// TwinCAT 3 PLC project plcProg
// ProgramVersion: 3.1.4024.0
// libraries:
//   Tc2_Standard, * (Beckhoff Automation GmbH)
//   Tc2_System, * (Beckhoff Automation GmbH)
//   Tc2_Utilities, * (Beckhoff Automation GmbH)
//   Tc3_Module, * (Beckhoff Automation GmbH)
//   VisuSymbols,3.5.10.0,System
// project tree:
//   DUTs/ E_EventType.TcDUT, E_OutputLevel.TcDUT, E_Direction.TcDUT, ST_Event.TcDUT
//   / GlobalTextList.TcGTLO, PlcTask.TcTTO, Visualization Manager.TcVMO (not stored)
//   GVLs/ GVL.TcGVL, HMI.TcGVL
//   POUs/ GroupController.TcPOU, SequentialLightSwitch.TcPOU, MAIN.TcPOU, ShutterSwitch.TcPOU, SimpleButton.TcPOU, UpStopDownButton.TcPOU
//   POUs/log_persistence/ EventLogger.TcPOU, FB_CsvPersistentEventStorage.TcPOU, F_UpdateEventTimestampWithSystemTime.TcPOU, I_PersistentEventStorage.TcIO (not stored)
//   VISUs/ Screen1.TcVIS
// real-time tasks:
//   TASK PlcTask: cycle T#10ms, priority 20, ADS port 350
// I/O:
//   DEVICE Device 1 (Beckhoff CCAT)
//   DEVICE Device 2 (CX-BK)
//     Box 1 (CX-BK)
// variable links:
//   plcProg/plcProg Instance <-> Device 2 (CX-BK)/Box 1 (CX-BK)
//     PlcTask Inputs/GVL.din_01zModulu3_przewod_14_s_26_1_gabinetNajnizej_bialopomaranczowy <-> Term 4 (KL1809)/Channel 1/Input
//     PlcTask Inputs/GVL.din_01zModulu4_przewod_11_s_42_1_rodzicow_1z1_bialobrazowy <-> Term 5 (KL1809)/Channel 1/Input
//     PlcTask Inputs/GVL.din_02zModulu3_przewod_14_s_26_1_gabinet_2z2_niebieski <-> Term 4 (KL1809)/Channel 2/Input
//     PlcTask Inputs/GVL.din_02zModulu4_przewod_11_s_42_1_rodzicow_1z1_bialopomaranczowy <-> Term 5 (KL1809)/Channel 2/Input
//     PlcTask Inputs/GVL.din_03zModulu2_przewod_3_s_30_1_kuchnia_2z2_zielony <-> Term 3 (KL1809)/Channel 3/Input
//     PlcTask Inputs/GVL.din_03zModulu3_przewod_14_s_26_1_gabinet_1z2_pomaranczowy <-> Term 4 (KL1809)/Channel 3/Input
//     PlcTask Inputs/GVL.din_03zModulu4_przewod_11_s_42_1_rodzicow_1z2_bialoniebieski <-> Term 5 (KL1809)/Channel 3/Input
//     PlcTask Inputs/GVL.din_04zModulu1_przewod_5_s_27_1_pralnia_2z2_niebieski <-> Term 2 (KL1809)/Channel 4/Input
//     PlcTask Inputs/GVL.din_04zModulu2_przewod_3_s_30_1_kuchnia_1z2_niebieski <-> Term 3 (KL1809)/Channel 4/Input
//     PlcTask Inputs/GVL.din_04zModulu3_przewod_14_s_40_1_lazienka_1z2_zielony <-> Term 4 (KL1809)/Channel 4/Input
//     PlcTask Inputs/GVL.din_05zModulu1_przewod_5_s_27_1_pralnia_1z2_pomaranczowy <-> Term 2 (KL1809)/Channel 5/Input
//     PlcTask Inputs/GVL.din_05zModulu2_przewod_3_s_30_1_kuchnia_2z2_pomaranczowy <-> Term 3 (KL1809)/Channel 5/Input
//     PlcTask Inputs/GVL.din_05zModulu3_przewod_14_s_40_1_lazienka_2z2_niebieski <-> Term 4 (KL1809)/Channel 5/Input
//     PlcTask Inputs/GVL.din_06zModulu1_przewod_1_s_25_1_koniecPrzedpokoju_2z2_zielony <-> Term 2 (KL1809)/Channel 6/Input
//     PlcTask Inputs/GVL.din_06zModulu2_przewod_3_s_30_1_kuchnia_1z2_brazowy <-> Term 3 (KL1809)/Channel 6/Input
//     PlcTask Inputs/GVL.din_07zModulu1_przewod_1_s_5_1_przedpokojPrzyDrzwiach_1z3_niebieski <-> Term 2 (KL1809)/Channel 7/Input
//     PlcTask Inputs/GVL.din_07zModulu2_przewod_3_s_30_1_kuchnia_2z2_bialoniebieski <-> Term 3 (KL1809)/Channel 7/Input
//     PlcTask Inputs/GVL.din_07zModulu3_przewod_5_s_23_1_pralniaNajnizej_niebieski <-> Term 4 (KL1809)/Channel 7/Input
//     PlcTask Inputs/GVL.din_08zModulu1_przewod_1_s_5_1_przedpokojPrzyDrzwiach_2z3_pomaranczowy <-> Term 2 (KL1809)/Channel 8/Input
//     PlcTask Inputs/GVL.din_08zModulu2_przewod_3_s_30_1_kuchnia_1z2_bialopomaranczowy <-> Term 3 (KL1809)/Channel 8/Input
//     PlcTask Inputs/GVL.din_08zModulu3_przewod_13_s_48_1_bezBalkonu_1z2_brazowy <-> Term 4 (KL1809)/Channel 8/Input
//     PlcTask Inputs/GVL.din_09zModulu1_przewod_1_s_5_1_przedpokojPrzyDrzwiach_3z3_brazowy <-> Term 2 (KL1809)/Channel 9/Input
//     PlcTask Inputs/GVL.din_09zModulu3_przewod_13_s_48_1_bezBalkonu_2z2_pomaranczowy <-> Term 4 (KL1809)/Channel 9/Input
//     PlcTask Inputs/GVL.din_10zModulu1_przewod_1_s_25_1_koniecPrzedpokojuElektronicznyPoczworny_1z4_brazowy <-> Term 2 (KL1809)/Channel 10/Input
//     PlcTask Inputs/GVL.din_10zModulu3_przewod_13_s_44_1_bezBalkonu_niebieski <-> Term 4 (KL1809)/Channel 10/Input
//     PlcTask Inputs/GVL.din_11zModulu1_przewod_1_s_25_1_koniecPrzedpokojuElektronicznyPoczworny_2z4_bialoniebieski <-> Term 2 (KL1809)/Channel 11/Input
//     PlcTask Inputs/GVL.din_11zModulu3_przewod_12_s_50_1_zBalkonem_1z2_brazowy <-> Term 4 (KL1809)/Channel 11/Input
//     PlcTask Inputs/GVL.din_12zModulu1_przewod_1_s_25_1_koniecPrzedpokojuElektronicznyPoczworny_3z4_bialopomaranczowy <-> Term 2 (KL1809)/Channel 12/Input
//     PlcTask Inputs/GVL.din_12zModulu2_przewod_4_s_14_1_dolSchodow_2z4_niebieski <-> Term 3 (KL1809)/Channel 12/Input
//     PlcTask Inputs/GVL.din_12zModulu3_przewod_12_s_50_1_zBalkonem_2z2_pomaranczowy <-> Term 4 (KL1809)/Channel 12/Input
//     PlcTask Inputs/GVL.din_13zModulu1_przewod_1_s_25_1_koniecPrzedpokojuElektronicznyPoczworny_4z4_bialobrazowy <-> Term 2 (KL1809)/Channel 13/Input
//     PlcTask Inputs/GVL.din_13zModulu2_przewod_4_s_14_1_dolSchodow_4z4_bialopomaranczowy <-> Term 3 (KL1809)/Channel 13/Input
//     PlcTask Inputs/GVL.din_13zModulu3_przewod_18_s_55_1_korytarzPrzySypialniach_1z1_zielony <-> Term 4 (KL1809)/Channel 13/Input
//     PlcTask Inputs/GVL.din_14ZModulu3_przewod_11_S_42_1_rodzicow_1z2_brazowy <-> Term 4 (KL1809)/Channel 14/Input
//     PlcTask Inputs/GVL.din_14zModulu1_przewod_4_s_21_1_slupekKuchnia_4z4_brazowy <-> Term 2 (KL1809)/Channel 14/Input
//     PlcTask Inputs/GVL.din_14zModulu2_przewod_18_s_38_1_goraSchodow_2z4_pomaranczowy <-> Term 3 (KL1809)/Channel 14/Input
//     PlcTask Inputs/GVL.din_15ZModulu3_przewod_11_S_42_1_rodzicow_2z2_pomaranczowy <-> Term 4 (KL1809)/Channel 15/Input
//     PlcTask Inputs/GVL.din_15zModulu1_przewod_4_s_21_1_slupekKuchnia_1z4_pomaranczowy <-> Term 2 (KL1809)/Channel 15/Input
//     PlcTask Inputs/GVL.din_15zModulu2_przewod_18_s_38_1_goraSchodow_3z4_brazowy <-> Term 3 (KL1809)/Channel 15/Input
//     PlcTask Inputs/GVL.din_16zModulu1_przewod_4_s_21_1_slupekKuchnia_2z4_bialoniebieski <-> Term 2 (KL1809)/Channel 16/Input
//     PlcTask Inputs/GVL.din_16zModulu2_przewod_14_s_26_1_gabinetPrawieNajnizej_brazowy <-> Term 3 (KL1809)/Channel 16/Input
//     PlcTask Inputs/GVL.din_16zModulu3_przewod_11_s_42_1_rodzicow_2z2_niebieski <-> Term 4 (KL1809)/Channel 16/Input
//     PlcTask Inputs/GVL.din_1_1_1 <-> Term 2 (KL1809)/Channel 1/Input
//     PlcTask Inputs/GVL.din_1_2_2 <-> Term 2 (KL1809)/Channel 2/Input
//     PlcTask Outputs/GVL.dout_10_zaluzja_gabinet_w_dol <-> Term 13 (KL2809)/Channel 4/Output
//     PlcTask Outputs/GVL.dout_10zModulu1_przewod_3_o_3_1_swiatloKontuarKuchnia <-> Term 9 (KL2809)/Channel 10/Output
//     PlcTask Outputs/GVL.dout_10zModulu2_przewod_xxx_swiatloGornaLazienkaPodlogowe <-> Term 10 (KL2809)/Channel 10/Output
//     PlcTask Outputs/GVL.dout_11_zaluzja_balkon_w_gore <-> Term 13 (KL2809)/Channel 5/Output
//     PlcTask Outputs/GVL.dout_11zModulu1_przewod_3_o_2_1_swiatloKuchniaSufit <-> Term 9 (KL2809)/Channel 11/Output
//     PlcTask Outputs/GVL.dout_11zModulu2_przewod_13_o_19_1_swiatloSypialniaBezBalkonu <-> Term 10 (KL2809)/Channel 11/Output
//     PlcTask Outputs/GVL.dout_12_zaluzja_balkon_w_dol <-> Term 13 (KL2809)/Channel 6/Output
//     PlcTask Outputs/GVL.dout_12zModulu1_przewod_11_o_18_1_2_swiatloNiskiIWysokiSufitSypialniaRodzicow <-> Term 9 (KL2809)/Channel 12/Output
//     PlcTask Outputs/GVL.dout_13_zaluzja_nad_wykuszem_w_gore <-> Term 13 (KL2809)/Channel 7/Output
//     PlcTask Outputs/GVL.dout_13zModulu1_przewod_4_o_10_1_swiatloGabinet <-> Term 9 (KL2809)/Channel 13/Output
//     PlcTask Outputs/GVL.dout_14_zaluzja_nad_wykuszem_w_dol <-> Term 13 (KL2809)/Channel 8/Output
//     PlcTask Outputs/GVL.dout_14zModulu1_przewod_14_o_24_1_3_swiatloWiszaceGornaLazienka <-> Term 9 (KL2809)/Channel 14/Output
//     PlcTask Outputs/GVL.dout_15_zaluzja_okno_bez_balkonu_w_gore <-> Term 13 (KL2809)/Channel 9/Output
//     PlcTask Outputs/GVL.dout_15zModulu1_przewod_18_o_18_1_2_swiatloKorytarzPunktySufit <-> Term 9 (KL2809)/Channel 15/Output
//     PlcTask Outputs/GVL.dout_16_zaluzja_okno_bez_balkonu_w_dol <-> Term 13 (KL2809)/Channel 10/Output
//     PlcTask Outputs/GVL.dout_16zModulu1_przewod_18_o_18_1_3_swiatloZyrandolKorytarz <-> Term 9 (KL2809)/Channel 16/Output
//     PlcTask Outputs/GVL.dout_1_zaluzja_pralnia_w_gore <-> Term 12 (KL2809)/Channel 11/Output
//     PlcTask Outputs/GVL.dout_1zModulu1_przewod_2_o_4_1_swiatloSalonJadalniaSufit <-> Term 9 (KL2809)/Channel 1/Output
//     PlcTask Outputs/GVL.dout_1zModulu2_przewod_1_s_70_1_swiatloPrzedpokojBlizejSalonu <-> Term 10 (KL2809)/Channel 1/Output
//     PlcTask Outputs/GVL.dout_2_zaluzja_pralnia_w_dol <-> Term 12 (KL2809)/Channel 12/Output
//     PlcTask Outputs/GVL.dout_2zModulu1_przewod_2_o_5_1_swiatloSalonKanapaSufit <-> Term 9 (KL2809)/Channel 2/Output
//     PlcTask Outputs/GVL.dout_2zModulu2_przewod_11_o_17_1_swiatloNadLozkiemSypialniaRodzicow <-> Term 10 (KL2809)/Channel 2/Output
//     PlcTask Outputs/GVL.dout_3_zaluzja_okno_narozne_kuchnia_w_gore <-> Term 12 (KL2809)/Channel 13/Output
//     PlcTask Outputs/GVL.dout_3zModulu1_przewod_2_o_7_1_swiatloPrzejscieZPrzedpokojuDoSalonuSufit <-> Term 9 (KL2809)/Channel 3/Output
//     PlcTask Outputs/GVL.dout_3zModulu2_przewod_14_o_23_1_3_swiatloSlabeGornaLazienka <-> Term 10 (KL2809)/Channel 3/Output
//     PlcTask Outputs/GVL.dout_4_zaluzja_okno_narozne_kuchnia_w_dol <-> Term 12 (KL2809)/Channel 14/Output
//     PlcTask Outputs/GVL.dout_4zModulu2_przewod_14_o_24_1_2_swiatloSrednieGornaLazienka <-> Term 10 (KL2809)/Channel 4/Output
//     PlcTask Outputs/GVL.dout_5_zaluzja_wykusz_w_gore <-> Term 12 (KL2809)/Channel 15/Output
//     PlcTask Outputs/GVL.dout_5zModulu2_przewod_14_o_23_1_2_swiatloMocneGornaLazienka <-> Term 10 (KL2809)/Channel 5/Output
//     PlcTask Outputs/GVL.dout_6_zaluzja_wykusz_w_dol <-> Term 12 (KL2809)/Channel 16/Output
//     PlcTask Outputs/GVL.dout_6zModulu1_przewod_podbitki <-> Term 9 (KL2809)/Channel 6/Output
//     PlcTask Outputs/GVL.dout_6zModulu2_przewod_3_o_1_1_swiatloKuchniaPodSzafkami <-> Term 10 (KL2809)/Channel 6/Output
//     PlcTask Outputs/GVL.dout_7_zaluzja_slide_w_gore <-> Term 13 (KL2809)/Channel 1/Output
//     PlcTask Outputs/GVL.dout_7zModulu1_przewod_1_o_27_1_swiatloPrzedpokojBlizejDrzwi <-> Term 9 (KL2809)/Channel 7/Output
//     PlcTask Outputs/GVL.dout_7zModulu2_przewod_xxxxxx_swiatloTrepy <-> Term 10 (KL2809)/Channel 7/Output
//     PlcTask Outputs/GVL.dout_8_zaluzja_slide_w_dol <-> Term 13 (KL2809)/Channel 2/Output
//     PlcTask Outputs/GVL.dout_8zModulu1_przewod_11_o_18_1_3_swiatloToaletkaSypialniaRodzicow <-> Term 9 (KL2809)/Channel 8/Output
//     PlcTask Outputs/GVL.dout_8zModulu2_przewod_18_o_14_1_swiatloKorytarzPrzypodlogowe <-> Term 10 (KL2809)/Channel 8/Output
//     PlcTask Outputs/GVL.dout_9_zaluzja_gabinet_w_gore <-> Term 13 (KL2809)/Channel 3/Output
//     PlcTask Outputs/GVL.dout_9zModulu1_przewod_5_o_11_1_swiatloPralnia <-> Term 9 (KL2809)/Channel 9/Output

CONFIGURATION plcProg
    RESOURCE PLC ON TwinCAT3
        TASK PlcTask(INTERVAL := T#10ms, PRIORITY := 20);
        PROGRAM MAIN WITH PlcTask : MAIN;
    END_RESOURCE
END_CONFIGURATION

// ---- DUTs/E_EventType.TcDUT
{attribute 'qualified_only'}
{attribute 'strict'}
{attribute 'to_string'}
TYPE E_EventType :
(
	Alarm := 0,
	Message := 1
);
END_TYPE

// ---- DUTs/E_OutputLevel.TcDUT
{attribute 'qualified_only'}
{attribute 'strict'}
{attribute 'to_string'}
TYPE E_OutputLevel :
(
	SMALL := 1,
	MEDIUM := 2,
	BIG := 3,
	SUPERSTRONG := 4	
);
END_TYPE

// ---- DUTs/E_Direction.TcDUT
{attribute 'qualified_only'}
{attribute 'strict'}
{attribute 'to_string'}
TYPE E_Direction :
(
	STOP := 0,
	UP := 1,
	DOWN := 2
);
END_TYPE

// ---- DUTs/ST_Event.TcDUT
TYPE ST_Event :
STRUCT
	eEventType : E_EventType;
	eEventSeverity : TcEventSeverity;
	nEventIdentity : UDINT;
	sEventText : STRING(255);
	dtTimestamp : DATE_AND_TIME;
END_STRUCT
END_TYPE

// ---- GVLs/GVL.TcGVL
{attribute 'qualified_only'}
VAR_GLOBAL CONSTANT
    MAX_SHUTTER_OUTPUTS : INT := 1;
	MAX_LIGHT_OUTPUTS_PER_LEVEL : INT := 3;
	MAX_SIMPLE_OUTPUTS : INT := 3;
	
	MAX_SHUTTERS : INT := 11;
	MAX_SEQUENTIAL_SWITCHES : INT := 0;//TODO 50 ALBO MNIEJ;
	MAX_SIMPLE_BUTTONS : INT := 18; //TODO PEWNIE WIECEJ
END_VAR

VAR_GLOBAL
	
	din_1_1_1 AT %I* : BOOL; //garaż po prawej stronie od drzwi
	din_1_2_2 AT %I* : BOOL; //garaż po lewej stronie od drzwi (wh-gn->bl) + pralnia po lewej stronie od drzwi, pierwszy od dołu (trzeba namierzyć)
	din_1_3_3 AT %I* : BOOL; //pralnia po lewej stronie od drzwi, drugi od dołu (trzeba namierzyć)
	din_1_4_4 AT %I* : BOOL; 
	din_1_5_5 AT %I* : BOOL;
	din_1_6_6 AT %I* : BOOL; 
	din_1_7_7 AT %I* : BOOL;
	din_1_8_8 AT %I* : BOOL;
	din_1_9_9 AT %I* : BOOL; 
	
	din_04zModulu1_przewod_5_s_27_1_pralnia_2z2_niebieski AT %I* : BOOL; //zasilanie bialo-zielony: Wlacznik roletowy w pralni dol
	din_05zModulu1_przewod_5_s_27_1_pralnia_1z2_pomaranczowy AT %I* : BOOL; //zasilanie bialo-zielony: Wlacznik roletowy w pralni gora
	din_06zModulu1_przewod_1_s_25_1_koniecPrzedpokoju_2z2_zielony AT %I* : BOOL; //zasilanie bialo-zielony: Wlacznik podwojny na koncu przedpokoju lub wlacznik poczworny na dole schodow 1/4
	din_07zModulu1_przewod_1_s_5_1_przedpokojPrzyDrzwiach_1z3_niebieski AT %I* : BOOL; //zasilanie bialo-zielony: Wlacznik swiatla w przedpokoju przy drzwiach 1/3
	din_08zModulu1_przewod_1_s_5_1_przedpokojPrzyDrzwiach_2z3_pomaranczowy AT %I* : BOOL; //zasilanie bialo-zielony: Wlacznik swiatla w przedpokoju przy drzwiach 2/3
	din_09zModulu1_przewod_1_s_5_1_przedpokojPrzyDrzwiach_3z3_brazowy AT %I* : BOOL; //zasilanie bialo-zielony: Wlacznik swiatla w przedpokoju przy drzwiach 3/3 lub wlacznik podwojny na koncu przedpokoju 1/2

	din_10zModulu1_przewod_1_s_25_1_koniecPrzedpokojuElektronicznyPoczworny_1z4_brazowy AT %I* : BOOL;//bylo din1_10_10 //zasilanie biało-zielony: Elektroniczny wlacznik swiatla w przedpokoju 1/4 lub wlacznik poczworny w kuchni na slupku 1/4
	din_11zModulu1_przewod_1_s_25_1_koniecPrzedpokojuElektronicznyPoczworny_2z4_bialoniebieski AT %I* : BOOL; //bylo din1_11_11 //zasilanie biało-zielony: Elektroniczny wlacznik swiatla w przedpokoju 2/4
	din_12zModulu1_przewod_1_s_25_1_koniecPrzedpokojuElektronicznyPoczworny_3z4_bialopomaranczowy AT %I* : BOOL; //bylo din1_12_12 //zasilanie biało-zielony: Elektroniczny wlacznik swiatla w przedpokoju 3/4 lub wlacznik poczworny na dole schodow 3/4
	din_13zModulu1_przewod_1_s_25_1_koniecPrzedpokojuElektronicznyPoczworny_4z4_bialobrazowy AT %I* : BOOL; //din_1_13_13 //zasilanie bialo-zielony: Elektroniczny wlacznik swiatla w przedpokoju 4/4	
	
	din_14zModulu1_przewod_4_s_21_1_slupekKuchnia_4z4_brazowy AT %I* : BOOL; //zasilanie bialo-zielony: Wlacznik poczworny w kuchni na slupku 4/4
	din_15zModulu1_przewod_4_s_21_1_slupekKuchnia_1z4_pomaranczowy AT %I* : BOOL; //zasilanie bialo-zielony: Wlacznik poczworny w kuchni na slupku 1/4
	din_16zModulu1_przewod_4_s_21_1_slupekKuchnia_2z4_bialoniebieski AT %I* : BOOL; //zasilanie bialo-zielony: Wlacznik poczworny w kuchni na slupku 2/4

	//todo swiatlo kontuar led, swiatlo zewnetrzne nad drzwiami
	din_03zModulu2_przewod_3_s_30_1_kuchnia_2z2_zielony AT %I* : BOOL; //zasilanie bialo-zielony: Wlacznik roletowy w kuchni kuchnia gora
    din_04zModulu2_przewod_3_s_30_1_kuchnia_1z2_niebieski AT %I* : BOOL; //zasilanie bialo-zielony: Wlacznik roletowy w kuchni kuchnia dol

	din_05zModulu2_przewod_3_s_30_1_kuchnia_2z2_pomaranczowy AT %I* : BOOL; //zasilanie bialo-zielony: Wlacznik roletowy w kuchni wykusz dol
	din_06zModulu2_przewod_3_s_30_1_kuchnia_1z2_brazowy AT %I* : BOOL; //zasilanie bialo-zielony: Wlacznik roletowy w kuchni wykusz gora

    din_07zModulu2_przewod_3_s_30_1_kuchnia_2z2_bialoniebieski AT %I* : BOOL; //zasilanie bialo-zielony: Wlacznik roletowy w kuchni slide dol
	din_08zModulu2_przewod_3_s_30_1_kuchnia_1z2_bialopomaranczowy AT %I* : BOOL; //zasilanie bialo-zielony: Wlacznik roletowy w kuchni slide gora
	
	din_12zModulu2_przewod_4_s_14_1_dolSchodow_2z4_niebieski AT %I* : BOOL; //zasilanie bialo-niebieski: Wlacznik poczworny na dole schodow 2/4
	din_13zModulu2_przewod_4_s_14_1_dolSchodow_4z4_bialopomaranczowy AT %I* : BOOL; //zasilanie bialo-niebieski: Wlacznik poczworny na dole schodow 4/4
	din_14zModulu2_przewod_18_s_38_1_goraSchodow_2z4_pomaranczowy AT %I* : BOOL; //zasilanie bialo-zielony: Wlacznik poczworny na gorze schodow 2/4
	din_15zModulu2_przewod_18_s_38_1_goraSchodow_3z4_brazowy AT %I* : BOOL; //zasilanie bialo-zielony: Wlacznik poczworny na gorze schodow 3/4

	din_16zModulu2_przewod_14_s_26_1_gabinetPrawieNajnizej_brazowy AT %I* : BOOL; //zasilanie bialo-zielony: Wlacznik w gabinecie prawie

	din_01zModulu3_przewod_14_s_26_1_gabinetNajnizej_bialopomaranczowy AT %I* : BOOL; //zasilanie bialo-zielony: Wlacznik w gabinecie najnizszy
	din_02zModulu3_przewod_14_s_26_1_gabinet_2z2_niebieski AT %I* : BOOL; //zasilanie bialo-zielony: Wlacznik roletowy w gabinecie dol
	din_03zModulu3_przewod_14_s_26_1_gabinet_1z2_pomaranczowy AT %I* : BOOL; //zasilanie bialo-zielony: Wlacznik roletowy w gabinecie gora
	
	din_04zModulu3_przewod_14_s_40_1_lazienka_1z2_zielony AT %I* : BOOL; //zasilanie bialo-zielony: Wlacznik podwojny w gornej lazience 1/2
	din_05zModulu3_przewod_14_s_40_1_lazienka_2z2_niebieski AT %I* : BOOL; //zasilanie bialo-zielony: Wlacznik podwojny w gornej lazience 2/2
	din_07zModulu3_przewod_5_s_23_1_pralniaNajnizej_niebieski AT %I* : BOOL; //zasilanie bialo-zielony: Wlacznik swiatla w pralni
	din_08zModulu3_przewod_13_s_48_1_bezBalkonu_1z2_brazowy AT %I* : BOOL; //zasilanie bialo-zielony: Wlacznik roletowy w sypialni bez balkonu 1/2
	din_09zModulu3_przewod_13_s_48_1_bezBalkonu_2z2_pomaranczowy AT %I* : BOOL; //zasilanie bialo-zielony: Wlacznik roletowy w sypialni bez balkonu 1/2
	
	din_10zModulu3_przewod_13_s_44_1_bezBalkonu_niebieski AT %I* : BOOL; //zasilanie bialo-zielony: Wlacznik swiatla w sypialni bez balkonu

	din_11zModulu3_przewod_12_s_50_1_zBalkonem_1z2_brazowy AT %I* : BOOL; //zasilanie bialo-zielony: Wlacznik roletowy w sypialni z balkonem gora
	din_12zModulu3_przewod_12_s_50_1_zBalkonem_2z2_pomaranczowy AT %I* : BOOL; //zasilanie bialo-zielony: Wlacznik roletowy w sypialni z balkonem dol
    
    din_13zModulu3_przewod_18_s_55_1_korytarzPrzySypialniach_1z1_zielony AT %I* : BOOL; //zasilanie bialo-zielony: Wylacznik swiatla korytarz przy sypialniach
	din_14ZModulu3_przewod_11_S_42_1_rodzicow_1z2_brazowy AT %I* : BOOL; //zasilanie bialo-zielony: Wlacznik roletowy w sypialni rodzicow gora
	din_15ZModulu3_przewod_11_S_42_1_rodzicow_2z2_pomaranczowy AT %I* : BOOL; //zasilanie bialo-zielony: Wlacznik roletowy w sypialni rodzicow dol
    din_16zModulu3_przewod_11_s_42_1_rodzicow_2z2_niebieski AT %I* : BOOL; //zasilanie bialo-zielony: Wlacznik swiatla w sypialni rodzicow przy drzwiach 2/2 lub wlacznik przy lozku po lewej 1/2 lub wlacznik przy lozku po prawej 1/2
	din_01zModulu4_przewod_11_s_42_1_rodzicow_1z1_bialobrazowy AT %I* : BOOL; //zasilanie bialo-zielony: Wlacznik swiatla w sypialni rodzicow przy drzwiach 1z1 lub wlacznik przy lozku po lewej 2/2 lub wlacznik przy lozku po prawej 2/2
    din_02zModulu4_przewod_11_s_42_1_rodzicow_1z1_bialopomaranczowy AT %I* : BOOL; //zasilanie bialo-zielony: Wlacznik swiatla w sypialni rodzicow przy drzwiach 1z1 lub wlacznik przy balkonie 1/1
	din_03zModulu4_przewod_11_s_42_1_rodzicow_1z2_bialoniebieski AT %I* : BOOL; //zasilanie bialo-zielony: Wlacznik swiatla w sypialni rodzicow przy drzwiach 1z2 lub wlacznik przy lozku po lewej 1/1 lub wlacznik przy lozku po prawej 1/1
	//todo wlacznik roletowy garaz
	
    din_1_14_14 AT %I* : BOOL;
	din_1_15_15 AT %I* : BOOL;
	din_1_16_16 AT %I* : BOOL;

	CsvPersistentEventStorage : FB_CsvPersistentEventStorage;
	EventLogger : EventLogger(CsvPersistentEventStorage);
	

//-------------------------------------------------------------------------------------------------	
//OUTPUTS
	dout_1_zaluzja_pralnia_w_gore AT %Q* : BOOL;
	douts_1_zaluzja_pralnia_w_gore : ARRAY[1..MAX_SHUTTER_OUTPUTS] OF BOOL; 	
	dout_2_zaluzja_pralnia_w_dol AT %Q* : BOOL;
	douts_2_zaluzja_pralnia_w_dol : ARRAY[1..MAX_SHUTTER_OUTPUTS] OF BOOL;
	
	dout_3_zaluzja_okno_narozne_kuchnia_w_gore AT %Q* : BOOL;
	douts_3_zaluzja_okno_narozne_kuchnia_w_gore : ARRAY[1..MAX_SHUTTER_OUTPUTS] OF BOOL;
	dout_4_zaluzja_okno_narozne_kuchnia_w_dol AT %Q* : BOOL;
	douts_4_zaluzja_okno_narozne_kuchnia_w_dol : ARRAY[1..MAX_SHUTTER_OUTPUTS] OF BOOL;
	
	dout_5_zaluzja_wykusz_w_gore AT %Q* : BOOL;	
	douts_5_zaluzja_wykusz_w_gore : ARRAY[1..MAX_SHUTTER_OUTPUTS] OF BOOL; 
	dout_6_zaluzja_wykusz_w_dol AT %Q* : BOOL;
	douts_6_zaluzja_wykusz_w_dol : ARRAY[1..MAX_SHUTTER_OUTPUTS] OF BOOL;
	
	dout_7_zaluzja_slide_w_gore AT %Q* : BOOL;	
	douts_7_zaluzja_slide_w_gore : ARRAY[1..MAX_SHUTTER_OUTPUTS] OF BOOL; 
	dout_8_zaluzja_slide_w_dol AT %Q* : BOOL;
	douts_8_zaluzja_slide_w_dol : ARRAY[1..MAX_SHUTTER_OUTPUTS] OF BOOL;
	
	dout_9_zaluzja_gabinet_w_gore AT %Q* : BOOL;	
	douts_9_zaluzja_gabinet_w_gore : ARRAY[1..MAX_SHUTTER_OUTPUTS] OF BOOL; 
	dout_10_zaluzja_gabinet_w_dol AT %Q* : BOOL;
	douts_10_zaluzja_gabinet_w_dol : ARRAY[1..MAX_SHUTTER_OUTPUTS] OF BOOL;
	
	dout_11_zaluzja_balkon_w_gore AT %Q* : BOOL;	
	douts_11_zaluzja_balkon_w_gore : ARRAY[1..MAX_SHUTTER_OUTPUTS] OF BOOL; 
	dout_12_zaluzja_balkon_w_dol AT %Q* : BOOL;	
	douts_12_zaluzja_balkon_w_dol : ARRAY[1..MAX_SHUTTER_OUTPUTS] OF BOOL; 
	
	dout_13_zaluzja_nad_wykuszem_w_gore AT %Q* : BOOL;
	douts_13_zaluzja_nad_wykuszem_w_gore : ARRAY[1..MAX_SHUTTER_OUTPUTS] OF BOOL;
	dout_14_zaluzja_nad_wykuszem_w_dol AT %Q* : BOOL;
	douts_14_zaluzja_nad_wykuszem_w_dol : ARRAY[1..MAX_SHUTTER_OUTPUTS] OF BOOL;
	
	dout_15_zaluzja_okno_bez_balkonu_w_gore AT %Q* : BOOL;	
	douts_15_zaluzja_okno_bez_balkonu_w_gore : ARRAY[1..MAX_SHUTTER_OUTPUTS] OF BOOL; 
	dout_16_zaluzja_okno_bez_balkonu_w_dol AT %Q* : BOOL;
	douts_16_zaluzja_okno_bez_balkonu_w_dol : ARRAY[1..MAX_SHUTTER_OUTPUTS] OF BOOL;
	
	dout_17_roleta_kotlownia_w_gore AT %Q* : BOOL;	
	douts_17_roleta_kotlownia_w_gore : ARRAY[1..MAX_SHUTTER_OUTPUTS] OF BOOL; 
	dout_18_roleta_kotlownia_w_dol AT %Q* : BOOL;
	douts_18_roleta_kotlownia_w_dol : ARRAY[1..MAX_SHUTTER_OUTPUTS] OF BOOL;
	
	dout_19_roleta_warsztat_w_gore AT %Q* : BOOL;	
	douts_19_roleta_warsztat_w_gore : ARRAY[1..MAX_SHUTTER_OUTPUTS] OF BOOL; 
	dout_20_roleta_warsztat_w_dol AT %Q* : BOOL;
	douts_20_roleta_warsztat_w_dol : ARRAY[1..MAX_SHUTTER_OUTPUTS] OF BOOL;
	
	dout_21_roleta_kotlownia_w_gore AT %Q* : BOOL;	
	douts_21_roleta_kotlownia_w_gore : ARRAY[1..MAX_SHUTTER_OUTPUTS] OF BOOL; 
	dout_22_roleta_kotlownia_w_dol AT %Q* : BOOL;
	douts_22_roleta_kotlownia_w_dol : ARRAY[1..MAX_SHUTTER_OUTPUTS] OF BOOL;
	
	

	dout_1zModulu1_przewod_2_o_4_1_swiatloSalonJadalniaSufit AT %Q* : BOOL; //2-o-4-1
		douts_swiatloSalonJadalniaSufit : ARRAY[1..MAX_LIGHT_OUTPUTS_PER_LEVEL] OF BOOL;
		
	dout_2zModulu1_przewod_2_o_5_1_swiatloSalonKanapaSufit AT %Q* : BOOL; //2-o-5-1
		douts_swiatloSalonKanapaSufit : ARRAY[1..MAX_LIGHT_OUTPUTS_PER_LEVEL] OF BOOL;
		
	dout_3zModulu1_przewod_2_o_7_1_swiatloPrzejscieZPrzedpokojuDoSalonuSufit AT %Q* : BOOL; //2-o-7-1
		douts_swiatloPrzejscieZPrzedpokojuDoSalonuSufit : ARRAY[1..MAX_LIGHT_OUTPUTS_PER_LEVEL] OF BOOL;
		
	dout_4zModulu1_przewod_2_o_6_1_swiatloSrodekSalonuSufit AT %Q* : BOOL; //2-o-6-1
		douts_swiatloSrodekSalonuSufit : ARRAY[1..MAX_LIGHT_OUTPUTS_PER_LEVEL] OF BOOL;
		
	dout_5zModulu1_przewod_swiatloPrzedDomem AT %Q* : BOOL; //frontowe pod balkonem
		douts_swiatloPrzedDomem : ARRAY[1..MAX_LIGHT_OUTPUTS_PER_LEVEL] OF BOOL;
		
	dout_6zModulu1_przewod_podbitki AT %Q* : BOOL; //podbitki
		douts_swiatloZewnetrznePodbitki : ARRAY[1..MAX_LIGHT_OUTPUTS_PER_LEVEL] OF BOOL;	
		
	dout_7zModulu1_przewod_1_o_27_1_swiatloPrzedpokojBlizejDrzwi AT %Q* : BOOL; //1_o_27_1
		douts_swiatloPrzedpokojBlizejDrzwi : ARRAY[1..MAX_LIGHT_OUTPUTS_PER_LEVEL] OF BOOL;
		
	dout_1zModulu2_przewod_1_s_70_1_swiatloPrzedpokojBlizejSalonu AT %Q* : BOOL; //1_s_70_1 to jest byly obwod 'S' sterowania 
		douts_swiatloPrzedpokojBlizejSalonu : ARRAY[1..MAX_LIGHT_OUTPUTS_PER_LEVEL] OF BOOL;
		
	dout_9zModulu1_przewod_5_o_11_1_swiatloPralnia AT %Q* : BOOL; //5_o_11_1
		douts_swiatloPralnia : ARRAY[1..MAX_LIGHT_OUTPUTS_PER_LEVEL] OF BOOL;
		
	dout_10zModulu1_przewod_3_o_3_1_swiatloKontuarKuchnia AT %Q* : BOOL; //3_o_3_1
		douts_swiatloKontuarKuchnia : ARRAY[1..MAX_LIGHT_OUTPUTS_PER_LEVEL] OF BOOL;
		
	dout_11zModulu1_przewod_3_o_2_1_swiatloKuchniaSufit AT %Q* : BOOL; //3_o_2_1
		douts_swiatloKuchniaSufit : ARRAY[1..MAX_LIGHT_OUTPUTS_PER_LEVEL] OF BOOL;
			
	dout_13zModulu1_przewod_4_o_10_1_swiatloGabinet AT %Q* : BOOL; //4_o_9_1, 4_o_10_1
		douts_swiatloGabinet : ARRAY[1..MAX_LIGHT_OUTPUTS_PER_LEVEL] OF BOOL;
		
	dout_15zModulu1_przewod_18_o_18_1_2_swiatloKorytarzPunktySufit AT %Q* : BOOL; //18_o_18_1 zasilanie z L
		douts_swiatloKorytarzPunktySufit : ARRAY[1..MAX_LIGHT_OUTPUTS_PER_LEVEL] OF BOOL;
		
	dout_16zModulu1_przewod_18_o_18_1_3_swiatloZyrandolKorytarz AT %Q* : BOOL; //18_o_18_1 zasilanie z PE
		douts_swiatloZyrandolKorytarz : ARRAY[1..MAX_LIGHT_OUTPUTS_PER_LEVEL] OF BOOL;

	dout_8zModulu1_przewod_11_o_18_1_3_swiatloToaletkaSypialniaRodzicow AT %Q* : BOOL; //11_o_18_1_3
		douts_swiatloToaletkaSypialniaRodzicow : ARRAY[1..MAX_LIGHT_OUTPUTS_PER_LEVEL] OF BOOL;
		
	dout_12zModulu1_przewod_11_o_18_1_2_swiatloNiskiIWysokiSufitSypialniaRodzicow AT %Q* : BOOL; //11_o_18_1_3
		douts_swiatloNiskiIWysokiSufitSypialniaRodzicow : ARRAY[1..MAX_LIGHT_OUTPUTS_PER_LEVEL] OF BOOL;
		
	dout_2zModulu2_przewod_11_o_17_1_swiatloNadLozkiemSypialniaRodzicow AT %Q* : BOOL; //11_o_17_1
		douts_swiatloNadLozkiemSypialniaRodzicow : ARRAY[1..MAX_LIGHT_OUTPUTS_PER_LEVEL] OF BOOL;
		
	dout_14zModulu1_przewod_14_o_24_1_3_swiatloWiszaceGornaLazienka AT %Q* : BOOL; //14_o_24_1_3
		douts_swiatloWiszaceGornaLazienka : ARRAY[1..MAX_LIGHT_OUTPUTS_PER_LEVEL] OF BOOL;
		
	dout_3zModulu2_przewod_14_o_23_1_3_swiatloSlabeGornaLazienka AT %Q* : BOOL; //14_o_23_1_3 
		douts_swiatloSlabeGornaLazienka : ARRAY[1..MAX_LIGHT_OUTPUTS_PER_LEVEL] OF BOOL;
		
	dout_4zModulu2_przewod_14_o_24_1_2_swiatloSrednieGornaLazienka AT %Q* : BOOL; //14_o_24_1_2 
		douts_swiatloSrednieGornaLazienka : ARRAY[1..MAX_LIGHT_OUTPUTS_PER_LEVEL] OF BOOL;
		
	dout_5zModulu2_przewod_14_o_23_1_2_swiatloMocneGornaLazienka AT %Q* : BOOL; //14_o_23_1_2 
		douts_swiatloMocneGornaLazienka : ARRAY[1..MAX_LIGHT_OUTPUTS_PER_LEVEL] OF BOOL;
		
	dout_6zModulu2_przewod_3_o_1_1_swiatloKuchniaPodSzafkami AT %Q* : BOOL; //3_o_1_1
		douts_swiatloKuchniaPodSzafkami : ARRAY[1..MAX_LIGHT_OUTPUTS_PER_LEVEL] OF BOOL;
	
	dout_7zModulu2_przewod_xxxxxx_swiatloTrepy AT %Q* : BOOL; //17-o-12-1,18-o-13-1
		douts_swiatloTrepy : ARRAY[1..MAX_LIGHT_OUTPUTS_PER_LEVEL] OF BOOL;
		
	dout_8zModulu2_przewod_18_o_14_1_swiatloKorytarzPrzypodlogowe AT %Q* : BOOL; //18-o-14-1
		douts_swiatloKorytarzPrzypodlogowe : ARRAY[1..MAX_LIGHT_OUTPUTS_PER_LEVEL] OF BOOL;
		
	dout_xxxxxxxx_przewod_xxxxxx_swiatloGaraz AT %Q* : BOOL; //xxxxx
		douts_swiatloGaraz : ARRAY[1..MAX_LIGHT_OUTPUTS_PER_LEVEL] OF BOOL;
		
	dout_10zModulu2_przewod_xxx_swiatloGornaLazienkaPodlogowe AT %Q* : BOOL;
		douts_swiatloGornaLazienkaWiszaceiPodlogowe : ARRAY[1..MAX_LIGHT_OUTPUTS_PER_LEVEL] OF BOOL;
	
	dout_11zModulu2_przewod_13_o_19_1_swiatloSypialniaBezBalkonu AT %Q* : BOOL; //13_o_19_1
		douts_swiatloSypialniaBezBalkonu : ARRAY[1..MAX_LIGHT_OUTPUTS_PER_LEVEL] OF BOOL;
END_VAR

// ---- GVLs/HMI.TcGVL
{attribute 'qualified_only'}
VAR_GLOBAL
	bStartPB : BOOL;
	bStopPB : BOOL;
	
	bStartTB : BOOL;
	bStopTB : BOOL;
	
	bIndicator1 : BOOL;
	bIndicator2 : BOOL;
	
	
	btn : BOOL;
	dayNightSwitch : BOOL;
		
	led1_1 : BOOL;
	led2_1 : BOOL;
	led2_2 : BOOL;
	led3 : BOOL;
	led4_1 : BOOL;
	led4_2 : BOOL;
	led4_3 : BOOL;
	//led4_4 : BOOL;
	
	
END_VAR

// ---- POUs/MAIN.TcPOU
PROGRAM MAIN
VAR
	initialized : BOOL := FALSE;
	serviceMode : BOOL := FALSE;
	stThisIsFirstInstanceOfAStructure : ST_Event;

	eEventType : E_EventType := E_EventType.Alarm;
	eEventSeverity : TcEventSeverity := TcEventSeverity.Info;
	nEventIdentity : UDINT := 44444;
	sEventText : STRING(255) := 'Some informational event';
	
	groupController : GroupController;

	wlaczniki_rolet_i_zaluzji : ARRAY[1..GVL.MAX_SHUTTERS] OF POINTER TO ShutterSwitch;
	wlacznik_1_zaluzja_pralnia : ShutterSwitch();
	wlacznik_2_zaluzje_kuchnia : ShutterSwitch();
	wlacznik_3_zaluzje_wykusz : ShutterSwitch();
	wlacznik_4_zaluzja_slide : ShutterSwitch();
    wlacznik_5_zaluzja_gabinet : ShutterSwitch();
    wlacznik_6_zaluzja_balkon : ShutterSwitch();
    wlacznik_7_zaluzja_nad_tarasem : ShutterSwitch();
	wlacznik_8_zaluzja_okno_bez_balkonu : ShutterSwitch();
	wlacznik_9_roleta_kotlownia : ShutterSwitch();
	wlacznik_10_roleta_warsztat : ShutterSwitch();
    wlacznik_11_rolety_garaz : ShutterSwitch();

	proste_wlaczniki_swiatel : ARRAY[1..GVL.MAX_SIMPLE_BUTTONS] OF POINTER TO SimpleButton;
		wlacznik_12_swiatlo_w_jadalni : SimpleButton();
		wlacznik_13_swiatlo_nad_kanapa_w_salonie : SimpleButton();
		wlacznik_14_swiatlo_w_przejsciu_z_przedpokoju_do_salonu : SimpleButton();
		wlacznik_15_swiatlo_na_srodku_salonu : SimpleButton(); //do namierzenia i podlaczenia
		wlacznik_16_swiatlo_nad_kontuarem_w_kuchni : SimpleButton(); //do namierzenia i podlaczenia
		wlacznik_17_swiatlo_w_kuchni_sufit : SimpleButton(); //do namierzenia i podlaczenia
		wlacznik_18_swiatlo_w_kuchni_pod_szafkami : SimpleButton(); //do namierzenia i podlaczenia jako 12V
		wlacznik_19_swiatlo_w_przedpokoju_blizej_salonu : SimpleButton(); //do namierzenia i podlaczenia
		wlacznik_20_swiatlo_w_przedpokoju_blizej_drzwi : SimpleButton(); //do namierzenia i podlaczenia
		wlacznik_21_swiatlo_pod_trepami : SimpleButton(); //do namierzenia i podlaczenia jako 12V albo 24V
		wlacznik_22_swiatlo_punkty_na_suficie_w_korytarzu : SimpleButton(); //do namierzenia i podlaczenia
		wlacznik_23_swiatlo_zyrandol_w_korytarzu : SimpleButton(); //do namierzenia i podlaczenia
		wlacznik_24_swiatlo_przypodlogowe_w_korytarzu : SimpleButton(); //do namierzenia i podlaczenia jako 12 V albo 24 V
		wlacznik_25_swiatlo_w_pralni : SimpleButton(); //do namierzenia i podlaczenia
		wlacznik_26_swiatlo_nad_toaletka_w_sypialni_rodzicow : SimpleButton(); //do namierzenia i podlaczenia
		wlacznik_27_swiatlo_niski_sufit_i_wysoki_sufit_w_sypialni_rodzicow : SimpleButton(); //do namierzenia i podlaczenia
		wlacznik_29_swiatlo_nad_lozkiem_w_sypialni_rodzicow : SimpleButton();//do namierzenia i podlaczenia
		wlacznik_30_swiatlo_frontowe : SimpleButton();//do namierzenia i podlaczenia
		wlacznik_31_swiatlo_podbitki : SimpleButton();
		wlacznik_32_swiatlo_w_garazu : SimpleButton();//do namierzenia i podlaczenia
		wlacznik_33_swiatlo_w_gabinecie : SimpleButton();
		wlacznik_34_swiatlo_w_sypialni_bez_balkonu : SimpleButton();
		wlacznik_35_swiatlo_w_gornej_lazience_wiszace : SimpleButton();
		
	sekwencyjne_wlaczniki_swiatel : ARRAY[1..GVL.MAX_SEQUENTIAL_SWITCHES] OF POINTER TO SequentialLightSwitch;
	(*	wlacznik_51_swiatlo_w_gornej_lazience_punkty_na_suficie_i_nocne : SequentialLightSwitch();
	*)
	wlaczniki_trojpozycyjne : ARRAY[1..10] OF UpStopDownButton;
		wlacznik_70_brama_garazowa : UpStopDownButton();//do namierzenia i podlaczenia
		
	isDay : BOOL := TRUE;
	minimumLogSeverity : TcEventSeverity := TcEventSeverity.Verbose;
END_VAR

VAR_IN_OUT

END_VAR

IF NOT initialized THEN
	systemService();
	IF serviceMode THEN
		JMP _programBypass;
	END_IF
	GVL.EventLogger.print1(level:=TcEventSeverity.Info, str1:='PLC started');
	
	//todo print date, all inputs and outputs values 
			//initButtons();	
	
	initializeButtons();
			F_UpdateEventTimestampWithSystemTime(stEvent := stThisIsFirstInstanceOfAStructure);	
			GVL.EventLogger.AddEvent(eEventType, eEventSeverity, nEventIdentity, sEventText);
			
	initialized := TRUE;
	groupController(shutters:= wlaczniki_rolet_i_zaluzji, 
					sequentialLightSwitches:= sekwencyjne_wlaczniki_swiatel,
					simpleButtons:= proste_wlaczniki_swiatel);

END_IF


//-------------------------------

//CsvPersistentEventStorage();


//buttontest.loop();

inputsOutputsLoop();
groupController.groupShutterLoop();


_programBypass :

METHOD initializeButtons
VAR_INPUT
END_VAR
// ShutterSwitch - pozostalo odkomentowac i podpiąć odpowiednie we/wy

wlacznik_1_zaluzja_pralnia(ID:=1, name:='Wlacznik zaluzji okna w pralni', 
		digitalInputUp:=GVL.din_05zModulu1_przewod_5_s_27_1_pralnia_1z2_pomaranczowy,
		digitalInputDown:=GVL.din_04zModulu1_przewod_5_s_27_1_pralnia_2z2_niebieski,
		up_outputs:=GVL.douts_1_zaluzja_pralnia_w_gore, 
		down_outputs:=GVL.douts_2_zaluzja_pralnia_w_dol, 
		shortTime:=T#500MS, longTime:= T#37S);
wlaczniki_rolet_i_zaluzji[1] := ADR(wlacznik_1_zaluzja_pralnia);

wlacznik_2_zaluzje_kuchnia(ID:=2, name:='Wlacznik zaluzji okna naroznego w kuchni', 
		digitalInputUp:=GVL.din_04zModulu2_przewod_3_s_30_1_kuchnia_1z2_niebieski,
		digitalInputDown:=GVL.din_03zModulu2_przewod_3_s_30_1_kuchnia_2z2_zielony,
		up_outputs:=GVL.douts_3_zaluzja_okno_narozne_kuchnia_w_gore, 
		down_outputs:=GVL.douts_4_zaluzja_okno_narozne_kuchnia_w_dol, 
		shortTime:=T#500MS, longTime:= T#37S);
wlaczniki_rolet_i_zaluzji[2] := ADR(wlacznik_2_zaluzje_kuchnia);

wlacznik_3_zaluzje_wykusz(ID:=3, name:='Wlacznik zaluzji przeszklenia wykuszu w salonie', 
		digitalInputUp:=GVL.din_06zModulu2_przewod_3_s_30_1_kuchnia_1z2_brazowy, 
		digitalInputDown:=GVL.din_05zModulu2_przewod_3_s_30_1_kuchnia_2z2_pomaranczowy,
		up_outputs:=GVL.douts_5_zaluzja_wykusz_w_gore, 
		down_outputs:=GVL.douts_6_zaluzja_wykusz_w_dol, 
		shortTime:=T#500MS, longTime:= T#56S);		
wlaczniki_rolet_i_zaluzji[3] := ADR(wlacznik_3_zaluzje_wykusz);

wlacznik_4_zaluzja_slide(ID:=4, name:='Wlacznik zaluzji drzwi slide na taras', 
		digitalInputUp:=GVL.din_08zModulu2_przewod_3_s_30_1_kuchnia_1z2_bialopomaranczowy, 
		digitalInputDown:=GVL.din_07zModulu2_przewod_3_s_30_1_kuchnia_2z2_bialoniebieski,
		up_outputs:=GVL.douts_7_zaluzja_slide_w_gore, 
		down_outputs:=GVL.douts_8_zaluzja_slide_w_dol, 
		shortTime:=T#500MS, longTime:= T#56S);				
wlaczniki_rolet_i_zaluzji[4] := ADR(wlacznik_4_zaluzja_slide);	

wlacznik_5_zaluzja_gabinet(ID:=5, name:='Wlacznik zaluzji okna w gabinecie', 
		digitalInputUp:=GVL.din_03zModulu3_przewod_14_s_26_1_gabinet_1z2_pomaranczowy,
		digitalInputDown:=GVL.din_02zModulu3_przewod_14_s_26_1_gabinet_2z2_niebieski,
		up_outputs:=GVL.douts_9_zaluzja_gabinet_w_gore, 
		down_outputs:=GVL.douts_10_zaluzja_gabinet_w_dol, 
		shortTime:=T#500MS, longTime:= T#37S);
wlaczniki_rolet_i_zaluzji[5] := ADR(wlacznik_5_zaluzja_gabinet);

wlacznik_6_zaluzja_balkon(ID:=6, name:='Wlacznik zaluzji drzwi sypialni z balkonem', 
		digitalInputUp:=GVL.din_11zModulu3_przewod_12_s_50_1_zBalkonem_1z2_brazowy,
		digitalInputDown:=GVL.din_12zModulu3_przewod_12_s_50_1_zBalkonem_2z2_pomaranczowy,
		up_outputs:=GVL.douts_11_zaluzja_balkon_w_gore, 
		down_outputs:=GVL.douts_12_zaluzja_balkon_w_dol, 
		shortTime:=T#500MS, longTime:= T#56S);
wlaczniki_rolet_i_zaluzji[6] := ADR(wlacznik_6_zaluzja_balkon);

wlacznik_7_zaluzja_nad_tarasem(ID:=7, name:='Wlacznik zaluzji drzwi w sypialni rodzicow', 
		digitalInputUp:=GVL.din_14ZModulu3_przewod_11_S_42_1_rodzicow_1z2_brazowy,
		digitalInputDown:=GVL.din_15ZModulu3_przewod_11_S_42_1_rodzicow_2z2_pomaranczowy,
		up_outputs:=GVL.douts_13_zaluzja_nad_wykuszem_w_gore, 
		down_outputs:=GVL.douts_14_zaluzja_nad_wykuszem_w_dol, 
		shortTime:=T#500MS, longTime:= T#56S);
wlaczniki_rolet_i_zaluzji[7] := ADR(wlacznik_7_zaluzja_nad_tarasem);

wlacznik_8_zaluzja_okno_bez_balkonu(ID:=8, name:='Wlacznik zaluzji okna w sypialni bez balkonu', 
		digitalInputUp:=GVL.din_08zModulu3_przewod_13_s_48_1_bezBalkonu_1z2_brazowy,
		digitalInputDown:=GVL.din_09zModulu3_przewod_13_s_48_1_bezBalkonu_2z2_pomaranczowy,
		up_outputs:=GVL.douts_15_zaluzja_okno_bez_balkonu_w_gore, 
		down_outputs:=GVL.douts_16_zaluzja_okno_bez_balkonu_w_dol, 
		shortTime:=T#500MS, longTime:= T#37S);
wlaczniki_rolet_i_zaluzji[8] := ADR(wlacznik_8_zaluzja_okno_bez_balkonu);
(*
wlacznik_9_roleta_kotlownia(ID:=9, name:='Wlacznik rolety okna w kotlowni', 
		digitalInputUp:=GVL.din_35,
		digitalInputDown:=GVL.din_36,
		up_outputs:=GVL.douts_17_roleta_kotlownia_w_gore, 
		down_outputs:=GVL.douts_18_roleta_kotlownia_w_dol, 
		shortTime:=T#250MS, longTime:= T#25S);
wlaczniki_rolet_i_zaluzji[9] := ADR(wlacznik_9_roleta_kotlownia);

wlacznik_10_roleta_warsztat(ID:=10, name:='Wlacznik rolety okna w warsztacie', 
		digitalInputUp:=GVL.din_37,
		digitalInputDown:=GVL.din_38,
		up_outputs:=GVL.douts_19_roleta_warsztat_w_gore, 
		down_outputs:=GVL.douts_20_roleta_warsztat_w_dol, 
		shortTime:=T#250MS, longTime:= T#25S);
wlaczniki_rolet_i_zaluzji[10] := ADR(wlacznik_10_roleta_warsztat);

wlacznik_11_rolety_garaz(ID:=11, name:='Wlacznik rolety okna w kotlowni', 
		digitalInputUp:=GVL.din_39,
		digitalInputDown:=GVL.din_40,
		up_outputs:=GVL.douts_21_roleta_kotlownia_w_gore, 
		down_outputs:=GVL.douts_22_roleta_kotlownia_w_dol, 
		shortTime:=T#250MS, longTime:= T#25S);
wlaczniki_rolet_i_zaluzji[11] := ADR(wlacznik_11_rolety_garaz);

*)

wlacznik_12_swiatlo_w_jadalni(ID:=12, name:='El. wl. sw. w przedpokoju 1/4 lub wl. sw. poczworny w kuchni na slupku 3/4',
		digitalInput:=GVL.din_10zModulu1_przewod_1_s_25_1_koniecPrzedpokojuElektronicznyPoczworny_1z4_brazowy, outputs:=GVL.douts_swiatloSalonJadalniaSufit,
        runAsYouPress:=FALSE, lightSwitch:= TRUE);		
proste_wlaczniki_swiatel[1] := ADR(wlacznik_12_swiatlo_w_jadalni);

wlacznik_13_swiatlo_nad_kanapa_w_salonie(ID:=13, name:='El. wl. swiatla w przedpokoju 2/4',
		digitalInput:=GVL.din_11zModulu1_przewod_1_s_25_1_koniecPrzedpokojuElektronicznyPoczworny_2z4_bialoniebieski, outputs:=GVL.douts_swiatloSalonKanapaSufit,
        runAsYouPress:=FALSE, lightSwitch:= TRUE);		
proste_wlaczniki_swiatel[2] := ADR(wlacznik_13_swiatlo_nad_kanapa_w_salonie);

wlacznik_14_swiatlo_w_przejsciu_z_przedpokoju_do_salonu(ID:=14, name:='El. wlacznik sw. w przedpokoju 3/4 lub wl. poczworny na dole schodow 1/4',
		digitalInput:=GVL.din_12zModulu1_przewod_1_s_25_1_koniecPrzedpokojuElektronicznyPoczworny_3z4_bialopomaranczowy, outputs:=GVL.douts_swiatloPrzejscieZPrzedpokojuDoSalonuSufit,
        runAsYouPress:=FALSE, lightSwitch:= TRUE);		
proste_wlaczniki_swiatel[3] := ADR(wlacznik_14_swiatlo_w_przejsciu_z_przedpokoju_do_salonu);

wlacznik_31_swiatlo_podbitki(ID:=31, name:='Wl. sw. w przedpokoju przy drzwiach 2/3',
		digitalInput:=GVL.din_08zModulu1_przewod_1_s_5_1_przedpokojPrzyDrzwiach_2z3_pomaranczowy, outputs:=GVL.douts_swiatloZewnetrznePodbitki,
        runAsYouPress:=FALSE, lightSwitch:= TRUE);		
proste_wlaczniki_swiatel[4] := ADR(wlacznik_31_swiatlo_podbitki);

wlacznik_17_swiatlo_w_kuchni_sufit(ID:=17, name:='Wl. sw. poczworny w kuchni na slupku 2/4',
		digitalInput:=GVL.din_16zModulu1_przewod_4_s_21_1_slupekKuchnia_2z4_bialoniebieski, outputs:=GVL.douts_swiatloKuchniaSufit,
        runAsYouPress:=FALSE, lightSwitch:= TRUE);		
proste_wlaczniki_swiatel[5] := ADR(wlacznik_17_swiatlo_w_kuchni_sufit);

wlacznik_16_swiatlo_nad_kontuarem_w_kuchni(ID:=16, name:='Wl. sw. poczworny w kuchni na slupku 1/4',
		digitalInput:=GVL.din_15zModulu1_przewod_4_s_21_1_slupekKuchnia_1z4_pomaranczowy, outputs:=GVL.douts_swiatloKontuarKuchnia,
        runAsYouPress:=FALSE, lightSwitch:= TRUE);	
proste_wlaczniki_swiatel[6] := ADR(wlacznik_16_swiatlo_nad_kontuarem_w_kuchni);

wlacznik_18_swiatlo_w_kuchni_pod_szafkami(ID:=18, name:='Wl. sw. poczworny w kuchni na slupku 4/4',
		digitalInput:=GVL.din_14zModulu1_przewod_4_s_21_1_slupekKuchnia_4z4_brazowy, outputs:=GVL.douts_swiatloKuchniaPodSzafkami,
        runAsYouPress:=FALSE, lightSwitch:= TRUE);	
proste_wlaczniki_swiatel[7] := ADR(wlacznik_18_swiatlo_w_kuchni_pod_szafkami);

wlacznik_33_swiatlo_w_gabinecie(ID:=33, name:='Wl. sw. w gabinecie najnizszy',
		digitalInput:=GVL.din_01zModulu3_przewod_14_s_26_1_gabinetNajnizej_bialopomaranczowy, outputs:=GVL.douts_swiatloGabinet,
        runAsYouPress:=FALSE, lightSwitch:= TRUE);	
proste_wlaczniki_swiatel[8] := ADR(wlacznik_33_swiatlo_w_gabinecie);

wlacznik_22_swiatlo_punkty_na_suficie_w_korytarzu(ID:=22, name:='Wl. sw. poczworny gora schodow 1/4',
		digitalInput:=GVL.din_12zModulu2_przewod_4_s_14_1_dolSchodow_2z4_niebieski, outputs:=GVL.douts_swiatloKorytarzPunktySufit,
        runAsYouPress:=FALSE, lightSwitch:= TRUE);	
proste_wlaczniki_swiatel[9] := ADR(wlacznik_22_swiatlo_punkty_na_suficie_w_korytarzu);

wlacznik_23_swiatlo_zyrandol_w_korytarzu(ID:=23, name:='Wl. sw. poczworny gora schodow 2/4',
		digitalInput:=GVL.din_14zModulu2_przewod_18_s_38_1_goraSchodow_2z4_pomaranczowy, outputs:=GVL.douts_swiatloZyrandolKorytarz,
        runAsYouPress:=FALSE, lightSwitch:= TRUE);	
proste_wlaczniki_swiatel[10] := ADR(wlacznik_23_swiatlo_zyrandol_w_korytarzu);

wlacznik_25_swiatlo_w_pralni(ID:=25, name:='Wl. sw. pralnia najnizszy',
		digitalInput:=GVL.din_07zModulu3_przewod_5_s_23_1_pralniaNajnizej_niebieski, outputs:=GVL.douts_swiatloPralnia,
        runAsYouPress:=FALSE, lightSwitch:= TRUE);	
proste_wlaczniki_swiatel[11] := ADR(wlacznik_25_swiatlo_w_pralni);

wlacznik_34_swiatlo_w_sypialni_bez_balkonu(ID:=34, name:='Wl. sw. sypialnia bez balkonu',
		digitalInput:=GVL.din_10zModulu3_przewod_13_s_44_1_bezBalkonu_niebieski, outputs:=GVL.douts_swiatloSypialniaBezBalkonu,
        runAsYouPress:=FALSE, lightSwitch:= TRUE);	
proste_wlaczniki_swiatel[12] := ADR(wlacznik_34_swiatlo_w_sypialni_bez_balkonu);

wlacznik_20_swiatlo_w_przedpokoju_blizej_drzwi(ID:=20, name:='Wl. sw. w przedpokoju przy drzwiach 3/3 lub na koncu przedpokoju 1/2',
		digitalInput:=GVL.din_09zModulu1_przewod_1_s_5_1_przedpokojPrzyDrzwiach_3z3_brazowy, outputs:=GVL.douts_swiatloPrzedpokojBlizejDrzwi,
        runAsYouPress:=FALSE, lightSwitch:= TRUE);	
proste_wlaczniki_swiatel[13] := ADR(wlacznik_20_swiatlo_w_przedpokoju_blizej_drzwi);

wlacznik_19_swiatlo_w_przedpokoju_blizej_salonu(ID:=19, name:='Wl. sw. na koncu przedpokoju 2/2',
		digitalInput:=GVL.din_06zModulu1_przewod_1_s_25_1_koniecPrzedpokoju_2z2_zielony, outputs:=GVL.douts_swiatloPrzedpokojBlizejSalonu,
        runAsYouPress:=FALSE, lightSwitch:= TRUE);	
proste_wlaczniki_swiatel[14] := ADR(wlacznik_19_swiatlo_w_przedpokoju_blizej_salonu);

wlacznik_26_swiatlo_nad_toaletka_w_sypialni_rodzicow(ID:=26, name:='Wl. sw. w sypialni rodzicow przy drzwiach 1/2 lub przy lozku 1/2',
		digitalInput:=GVL.din_16zModulu3_przewod_11_s_42_1_rodzicow_2z2_niebieski, outputs:=GVL.douts_swiatloToaletkaSypialniaRodzicow,
        runAsYouPress:=FALSE, lightSwitch:= TRUE);	
proste_wlaczniki_swiatel[15] := ADR(wlacznik_26_swiatlo_nad_toaletka_w_sypialni_rodzicow);

wlacznik_27_swiatlo_niski_sufit_i_wysoki_sufit_w_sypialni_rodzicow(ID:=27, name:='Wl. sw. w sypialni rodzicow przy drzwiach 1/1 lub przy lozku 2/2',
		digitalInput:=GVL.din_01zModulu4_przewod_11_s_42_1_rodzicow_1z1_bialobrazowy, outputs:=GVL.douts_swiatloNiskiIWysokiSufitSypialniaRodzicow,
        runAsYouPress:=FALSE, lightSwitch:= TRUE);	
proste_wlaczniki_swiatel[16] := ADR(wlacznik_27_swiatlo_niski_sufit_i_wysoki_sufit_w_sypialni_rodzicow);

wlacznik_29_swiatlo_nad_lozkiem_w_sypialni_rodzicow(ID:=29, name:='Wl. sw. w sypialni rodzicow przy drzwiach 1/2 lub przy lozku 1/1',
		digitalInput:=GVL.din_03zModulu4_przewod_11_s_42_1_rodzicow_1z2_bialoniebieski, outputs:=GVL.douts_swiatloNadLozkiemSypialniaRodzicow,
        runAsYouPress:=FALSE, lightSwitch:= TRUE);	
proste_wlaczniki_swiatel[17] := ADR(wlacznik_29_swiatlo_nad_lozkiem_w_sypialni_rodzicow);

wlacznik_35_swiatlo_w_gornej_lazience_wiszace(ID:=35, name:='Wl. sw. w gornej lazience 2/2 lub na korytarzu 2/2',
		digitalInput:=GVL.din_05zModulu3_przewod_14_s_40_1_lazienka_2z2_niebieski, outputs:=GVL.douts_swiatloWiszaceGornaLazienka,
        runAsYouPress:=FALSE, lightSwitch:= TRUE);	
proste_wlaczniki_swiatel[18] := ADR(wlacznik_35_swiatlo_w_gornej_lazience_wiszace);

(*
wlacznik_51_swiatlo_w_gornej_lazience_punkty_na_suficie_i_nocne(ID:= 51, name:='Smart wl. sw. w gornej lazience 1/2',
		digitalInput:=GVL.din_04zModulu3_przewod_14_s_40_1_lazienka_1z2_zielony, 
		small_outputs:=GVL.douts_swiatloSlabeGornaLazienka,
		medium_outputs:=GVL.douts_swiatloSrednieGornaLazienka,
		big_outputs:=GVL.douts_swiatloMocneGornaLazienka,
		superstrong_outputs:=GVL.douts_swiatloMocneGornaLazienka,
		defaultDayOutput:=E_OutputLevel.BIG,
		defaultNightOutput:=E_OutputLevel.SMALL,
		levelsManaged:=4);
sekwencyjne_wlaczniki_swiatel[1] := ADR(wlacznik_51_swiatlo_w_gornej_lazience_punkty_na_suficie_i_nocne);
*)

//prosteWlaczniki[1] := wlacznik_ogrzewania_lustra; 

//wlacznikiTrojpozycyjne[1] := wlacznik_bramy_garazowej;
END_METHOD

METHOD inputsOutputsLoop : BOOL
VAR_INPUT
END_VAR
//TODO pozamieniac dout_1_zaluzja_pralnia_w_gore na konkretny indeksowany DOUT


wlaczniki_rolet_i_zaluzji[1]^.loop();
	GVL.dout_1_zaluzja_pralnia_w_gore := GVL.douts_1_zaluzja_pralnia_w_gore[1];
	GVL.dout_2_zaluzja_pralnia_w_dol := GVL.douts_2_zaluzja_pralnia_w_dol[1];
 	
 wlaczniki_rolet_i_zaluzji[2]^.loop();
	GVL.dout_3_zaluzja_okno_narozne_kuchnia_w_gore := GVL.douts_3_zaluzja_okno_narozne_kuchnia_w_gore[1];
	GVL.dout_4_zaluzja_okno_narozne_kuchnia_w_dol := GVL.douts_4_zaluzja_okno_narozne_kuchnia_w_dol[1];
	
wlaczniki_rolet_i_zaluzji[3]^.loop();
	GVL.dout_5_zaluzja_wykusz_w_gore := GVL.douts_5_zaluzja_wykusz_w_gore[1];
	GVL.dout_6_zaluzja_wykusz_w_dol := GVL.douts_6_zaluzja_wykusz_w_dol[1];
	
wlaczniki_rolet_i_zaluzji[4]^.loop();
	GVL.dout_7_zaluzja_slide_w_gore := GVL.douts_7_zaluzja_slide_w_gore[1];
	GVL.dout_8_zaluzja_slide_w_dol := GVL.douts_8_zaluzja_slide_w_dol[1];

wlaczniki_rolet_i_zaluzji[5]^.loop();
	GVL.dout_9_zaluzja_gabinet_w_gore := GVL.douts_9_zaluzja_gabinet_w_gore[1];
	GVL.dout_10_zaluzja_gabinet_w_dol := GVL.douts_10_zaluzja_gabinet_w_dol[1];
	
wlaczniki_rolet_i_zaluzji[6]^.loop();
	GVL.dout_11_zaluzja_balkon_w_gore := GVL.douts_11_zaluzja_balkon_w_gore[1];
	GVL.dout_12_zaluzja_balkon_w_dol := GVL.douts_12_zaluzja_balkon_w_dol[1];
		
wlaczniki_rolet_i_zaluzji[7]^.loop();
	GVL.dout_13_zaluzja_nad_wykuszem_w_gore := GVL.douts_13_zaluzja_nad_wykuszem_w_gore[1];
	GVL.dout_14_zaluzja_nad_wykuszem_w_dol := GVL.douts_14_zaluzja_nad_wykuszem_w_dol[1];
	
wlaczniki_rolet_i_zaluzji[8]^.loop();
	GVL.dout_15_zaluzja_okno_bez_balkonu_w_gore := GVL.douts_15_zaluzja_okno_bez_balkonu_w_gore[1];
	GVL.dout_16_zaluzja_okno_bez_balkonu_w_dol := GVL.douts_16_zaluzja_okno_bez_balkonu_w_dol[1];

//TODO pozostale wlaczniki rolet


//wlaczniki_swiatel[1]^.loop();

//	GVL.b_led_2 := GVL.douts_ledy2[1];
//	GVL.b_led_3 := GVL.douts_ledy3[1];
	
//wlaczniki_swiatel[2]^.loop();
//	GVL.b_led_1 := GVL.douts_ledy1[1];

(*
sekwencyjne_wlaczniki_swiatel[1]^.loop();
	GVL.dout_3zModulu2_przewod_14_o_23_1_3_swiatloSlabeGornaLazienka := GVL.douts_swiatloSlabeGornaLazienka[1];
	GVL.dout_4zModulu2_przewod_14_o_24_1_2_swiatloSrednieGornaLazienka := GVL.douts_swiatloSrednieGornaLazienka[1];
	GVL.dout_5zModulu2_przewod_14_o_23_1_2_swiatloMocneGornaLazienka := GVL.douts_swiatloMocneGornaLazienka[1];
*)
	
proste_wlaczniki_swiatel[1]^.loop();
	GVL.dout_1zModulu1_przewod_2_o_4_1_swiatloSalonJadalniaSufit := GVL.douts_swiatloSalonJadalniaSufit[1];
	
proste_wlaczniki_swiatel[2]^.loop();
	GVL.dout_2zModulu1_przewod_2_o_5_1_swiatloSalonKanapaSufit := GVL.douts_swiatloSalonKanapaSufit[1];

proste_wlaczniki_swiatel[3]^.loop();
	GVL.dout_3zModulu1_przewod_2_o_7_1_swiatloPrzejscieZPrzedpokojuDoSalonuSufit := GVL.douts_swiatloPrzejscieZPrzedpokojuDoSalonuSufit[1];
	
proste_wlaczniki_swiatel[4]^.loop();
	GVL.dout_6zModulu1_przewod_podbitki := GVL.douts_swiatloZewnetrznePodbitki[1];

proste_wlaczniki_swiatel[5]^.loop();
	GVL.dout_11zModulu1_przewod_3_o_2_1_swiatloKuchniaSufit := GVL.douts_swiatloKuchniaSufit[1];
	
proste_wlaczniki_swiatel[6]^.loop();
	GVL.dout_10zModulu1_przewod_3_o_3_1_swiatloKontuarKuchnia := GVL.douts_swiatloKontuarKuchnia[1];	
	
proste_wlaczniki_swiatel[7]^.loop();
	GVL.dout_6zModulu2_przewod_3_o_1_1_swiatloKuchniaPodSzafkami := GVL.douts_swiatloKuchniaPodSzafkami[1];	
	
proste_wlaczniki_swiatel[8]^.loop();
	GVL.dout_13zModulu1_przewod_4_o_10_1_swiatloGabinet := GVL.douts_swiatloGabinet[1];	
	
proste_wlaczniki_swiatel[9]^.loop();
	GVL.dout_15zModulu1_przewod_18_o_18_1_2_swiatloKorytarzPunktySufit := GVL.douts_swiatloKorytarzPunktySufit[1];

proste_wlaczniki_swiatel[10]^.loop();
	GVL.dout_16zModulu1_przewod_18_o_18_1_3_swiatloZyrandolKorytarz := GVL.douts_swiatloZyrandolKorytarz[1];
	
proste_wlaczniki_swiatel[11]^.loop();
	GVL.dout_9zModulu1_przewod_5_o_11_1_swiatloPralnia := GVL.douts_swiatloPralnia[1];
	
proste_wlaczniki_swiatel[12]^.loop();
	GVL.dout_11zModulu2_przewod_13_o_19_1_swiatloSypialniaBezBalkonu := GVL.douts_swiatloSypialniaBezBalkonu[1];	
	
proste_wlaczniki_swiatel[13]^.loop();
	GVL.dout_7zModulu1_przewod_1_o_27_1_swiatloPrzedpokojBlizejDrzwi := GVL.douts_swiatloPrzedpokojBlizejDrzwi[1];	
	
proste_wlaczniki_swiatel[14]^.loop();
	GVL.dout_1zModulu2_przewod_1_s_70_1_swiatloPrzedpokojBlizejSalonu := GVL.douts_swiatloPrzedpokojBlizejSalonu[1];	
			
proste_wlaczniki_swiatel[15]^.loop();
	GVL.dout_8zModulu1_przewod_11_o_18_1_3_swiatloToaletkaSypialniaRodzicow := GVL.douts_swiatloToaletkaSypialniaRodzicow[1];	
	
proste_wlaczniki_swiatel[16]^.loop();
	GVL.dout_12zModulu1_przewod_11_o_18_1_2_swiatloNiskiIWysokiSufitSypialniaRodzicow := GVL.douts_swiatloNiskiIWysokiSufitSypialniaRodzicow[1];	
	
proste_wlaczniki_swiatel[17]^.loop();
	GVL.dout_2zModulu2_przewod_11_o_17_1_swiatloNadLozkiemSypialniaRodzicow := GVL.douts_swiatloNadLozkiemSypialniaRodzicow[1];	

proste_wlaczniki_swiatel[18]^.loop();
	GVL.dout_14zModulu1_przewod_14_o_24_1_3_swiatloWiszaceGornaLazienka := GVL.douts_swiatloWiszaceGornaLazienka[1];
END_METHOD

METHOD systemService
VAR_INPUT
END_VAR

VAR
	neededHigh : BOOL := FALSE;
	neededLow : BOOL := TRUE;
END_VAR
neededHigh := GVL.din_1_1_1;//_1;
neededLow := GVL.din_1_2_2;//_2;

IF serviceMode THEN
	JMP _wait_for_service_mode_exit;
END_IF

ADSLOGSTR(ADSLOG_MSGTYPE_ERROR, 'Device booted', '');
ADSLOGSTR(ADSLOG_MSGTYPE_ERROR, 'To enter service mode next time set DIGITAL INPUT 1 to TRUE and DIGITAL INPUT 2 to FALSE', '');
IF neededHigh AND NOT neededLow THEN
	ADSLOGSTR(ADSLOG_MSGTYPE_ERROR, 'Service mode entered', '');
	serviceMode := TRUE;
END_IF

_wait_for_service_mode_exit :

IF neededLow THEN
	ADSLOGSTR(ADSLOG_MSGTYPE_ERROR, 'Exiting service mode', '');
	serviceMode := FALSE;
END_IF
END_METHOD

END_PROGRAM

// ---- POUs/GroupController.TcPOU
FUNCTION_BLOCK GroupController
VAR CONSTANT
END_VAR
VAR_INPUT
	shutters : ARRAY[1..GVL.MAX_SHUTTERS] OF POINTER TO ShutterSwitch;
	sequentialLightSwitches : ARRAY[1..GVL.MAX_SEQUENTIAL_SWITCHES] OF POINTER TO SequentialLightSwitch;
	simpleButtons : ARRAY[1..GVL.MAX_SIMPLE_BUTTONS] OF POINTER TO SimpleButton;
END_VAR
VAR_OUTPUT
END_VAR
VAR
	shuttersCloseRequested : BOOL := FALSE;
	shuttersOpenRequested : BOOL := FALSE;
	
	shutterMoveInterval : TP := (PT := T#10S);
	currentShutterNumber : INT := 1;
END_VAR

METHOD PRIVATE getSource : STRING
VAR_INPUT
END_VAR

VAR
END_VAR
getSource := ' - Group controller';
END_METHOD

METHOD PUBLIC groupShutterLoop

VAR_INPUT
END_VAR

VAR

END_VAR
IF NOT shuttersCloseRequested THEN
	JMP _ret;
END_IF

shutterMoveInterval(IN:= FALSE);

IF NOT shutterMoveInterval.Q THEN
	GVL.EventLogger.print3(level:= TcEventSeverity.Verbose, str1:='Closing shutter number=', str2:= TO_STRING(currentShutterNumber), str3:=getSource());
	shutterMoveInterval(IN:= TRUE);
	shutters[currentShutterNumber]^.moveDownMax(requestedExternally:= TRUE);
	currentShutterNumber := currentShutterNumber + 1;
END_IF

IF currentShutterNumber > GVL.MAX_SHUTTERS THEN
	GVL.EventLogger.print3(level:= TcEventSeverity.Verbose, str1:='Closing shutters finished, closed=', str2:= TO_STRING(currentShutterNumber-1), str3:=getSource());
	shuttersCloseRequested := FALSE;
	currentShutterNumber := 1;
END_IF
 
_ret :


IF NOT shuttersOpenRequested THEN
	JMP _ret2;
END_IF

shutterMoveInterval(IN:= FALSE);

IF NOT shutterMoveInterval.Q THEN
	GVL.EventLogger.print3(level:= TcEventSeverity.Verbose, str1:='Opening shutter number=', str2:= TO_STRING(currentShutterNumber), str3:=getSource());
	shutterMoveInterval(IN:= TRUE);
	shutters[currentShutterNumber]^.moveUpMax(requestedExternally:= TRUE);
	currentShutterNumber := currentShutterNumber + 1;
END_IF

IF currentShutterNumber > GVL.MAX_SHUTTERS THEN
	GVL.EventLogger.print3(level:= TcEventSeverity.Verbose, str1:='Opening shutters finished, closed=', str2:= TO_STRING(currentShutterNumber), str3:=getSource());
	shuttersOpenRequested := FALSE;
	currentShutterNumber := 1;
END_IF

_ret2 :
END_METHOD

  METHOD requestLightsOff : BOOL
VAR_INPUT
END_VAR

VAR
	i : INT;

END_VAR
GVL.EventLogger.print3(level:= TcEventSeverity.Info, str1:='Lights OFF requested', str2:= '', str3:=getSource());

(*
FOR i := 1 TO GVL.MAX_SEQUENTIAL_SWITCHES BY 1 DO
	sequentialLightSwitches[i]^.turnOff();
END_FOR
*)
FOR i := 1 TO GVL.MAX_SIMPLE_BUTTONS BY 1 DO
	IF simpleButtons[i]^.isLightSwitch() THEN
		simpleButtons[i]^.turnOff();
	END_IF
END_FOR
END_METHOD

METHOD requestLightsOnDefault : BOOL
VAR_INPUT
END_VAR

VAR
	i : INT;
END_VAR
GVL.EventLogger.print3(level:= TcEventSeverity.Info, str1:='Lights ON default requested', str2:= '', str3:=getSource());

(*
FOR i := 1 TO GVL.MAX_SEQUENTIAL_SWITCHES BY 1 DO
	sequentialLightSwitches[i]^.turnOnDefault();
END_FOR
*)
FOR i := 1 TO GVL.MAX_SIMPLE_BUTTONS BY 1 DO
	IF simpleButtons[i]^.isLightSwitch() THEN
		simpleButtons[i]^.turnOn();
	END_IF
END_FOR
END_METHOD

METHOD PUBLIC requestShuttersClose : BOOL
VAR_INPUT
END_VAR
GVL.EventLogger.print3(level:= TcEventSeverity.Info, str1:='Shutters CLOSE requested', str2:= '', str3:=getSource());

shuttersCloseRequested := TRUE;
shuttersOpenRequested := FALSE;
currentShutterNumber := 1;
END_METHOD

METHOD PUBLIC requestShuttersOpen : BOOL
VAR_INPUT
END_VAR
GVL.EventLogger.print3(level:= TcEventSeverity.Info, str1:='Shutters OPEN requested', str2:= '', str3:=getSource());

shuttersOpenRequested := TRUE;
shuttersCloseRequested := FALSE;
currentShutterNumber := 1;
END_METHOD

END_FUNCTION_BLOCK

// ---- POUs/ShutterSwitch.TcPOU
FUNCTION_BLOCK ShutterSwitch

VAR CONSTANT
	MAX_OUTPUTS_PER_LEVEL : INT := GVL.MAX_SHUTTER_OUTPUTS;
END_VAR

VAR_INPUT
	ID : INT;
	name : STRING := 'Shutter switch';
	digitalInputUp : REFERENCE TO BOOL;
	digitalInputDown : REFERENCE TO BOOL;
	
	up_outputs : REFERENCE TO ARRAY[1..MAX_OUTPUTS_PER_LEVEL] OF BOOL;
	down_outputs : REFERENCE TO ARRAY[1..MAX_OUTPUTS_PER_LEVEL] OF BOOL;
	
	shortTime : TIME := T#250MS;
	longTime : TIME := T#60S;
END_VAR

VAR_OUTPUT
END_VAR

VAR
	initialized : BOOL := FALSE;
	canPrintGoUp : BOOL := TRUE;
	canPrintGoDown : BOOL := TRUE;
	longMoveAborted : BOOL := FALSE;
	justStopped : BOOL := FALSE;
	requestedByGroupController : BOOL := FALSE;
	
	isClosing : BOOL := FALSE;
	isOpening : BOOL := FALSE;
	
    pressedUp : R_TRIG;
	pressedDown : R_TRIG;
	releasedUp : F_TRIG;
	releasedDown : F_TRIG;
	
	pressedUpTimer : TON := (PT := T#10S);	
	pressedDownTimer : TON := (PT := T#10S);
	
	shortDistanceUp : TP := (PT := shortTime);
	longDistanceUp : TP := (PT := longTime);
	shortDistanceDown : TP := (PT := shortTime);
	longDistanceDown : TP := (PT := longTime);
	
	shutterCooldownTimer : TP := (PT := T#1500MS);
	
	pressedUpMiliseconds : INT := 0;
	pressedDownMiliseconds : INT := 0;	
	
	goUpRequested : BOOL := FALSE;
	goDownRequested : BOOL := FALSE;
	
	manualControl : BOOL := FALSE;
	inactivityTimeout : TP := (PT := T#1100MS);
	consecutiveClicks : INT := 0;
END_VAR

IF NOT initialized THEN
	initialized := TRUE;	
END_IF

shortDistanceUp(PT := shortTime);
longDistanceUp(PT := longTime);
shortDistanceDown(PT := shortTime);
longDistanceDown(PT := longTime);

METHOD PRIVATE calculatePressedTimeMiliseconds
VAR_INPUT
END_VAR
//long hold up
IF digitalInputUp AND TIME_TO_INT(pressedUpTimer.ET) <> 0 THEN
	pressedUpMiliseconds := TIME_TO_INT(pressedUpTimer.ET);
END_IF

//long hold down
IF digitalInputDown AND TIME_TO_INT(pressedDownTimer.ET) <> 0 THEN
	pressedDownMiliseconds := TIME_TO_INT(pressedDownTimer.ET);
END_IF
END_METHOD

METHOD doSpecialAction : BOOL
VAR_INPUT
END_VAR

VAR
	i: INT;
END_VAR
CASE ID OF
	//TODO pamietac
//	3:
//		GVL.EventLogger.print3(level:=TcEventSeverity.Info, str1:='Special action for button 1 - ', str2:='turning off all lights', str3:=getSource());
//		MAIN.groupController.requestLightsOff();
		
	2:
		GVL.EventLogger.print3(level:=TcEventSeverity.Info, str1:='Special action for button 2 - ', str2:='opening all shutters', str3:=getSource());
		MAIN.groupController.requestShuttersOpen();
		
	4:
		GVL.EventLogger.print3(level:=TcEventSeverity.Info, str1:='Special action for button 4 - ', str2:='closing all shutters', str3:=getSource());
		MAIN.groupController.requestShuttersClose();
		
END_CASE
END_METHOD

METHOD PRIVATE getSource : STRING(255)
VAR_INPUT
END_VAR

VAR
	details : STRING(255);
END_VAR
details := CONCAT(STR1:=' - shutter switch, ID: ', STR2:=TO_STRING(ID));
details := CONCAT(STR1:=details, STR2:=', digital input up: ');
details := CONCAT(STR1:=details, STR2:=TO_STRING(digitalInputUp));
details := CONCAT(STR1:=details, STR2:=', digital input down: ');
details := CONCAT(STR1:=details, STR2:=TO_STRING(digitalInputDown));
details := CONCAT(STR1:=details, STR2:=', request by group controller: ');
details := CONCAT(STR1:=details, STR2:=TO_STRING(requestedByGroupController));
details := CONCAT(STR1:=details, STR2:=', name: ');
details := CONCAT(STR1:=details, STR2:=name);

getSource := details;
END_METHOD

METHOD PRIVATE inputsOutputsLoop
VAR_INPUT
END_VAR
pressedUp(CLK:= digitalInputUp);
pressedDown(CLK:= digitalInputDown);
releasedUp(CLK:= digitalInputUp);
releasedDown(CLK:= digitalInputDown);
pressedUpTimer(IN := digitalInputUp);
pressedDownTimer(IN := digitalInputDown);
shortDistanceDown(IN:=FALSE);
longDistanceDown(IN:=FALSE);
shortDistanceUp(IN:=FALSE);
longDistanceUp(IN:=FALSE);
inactivityTimeout(IN:= FALSE);
END_METHOD

METHOD loop : BOOL
VAR_INPUT
END_VAR

VAR
END_VAR
inputsOutputsLoop();	
		
onAnyPressedDown();

//prevent both pressed
IF digitalInputUp AND digitalInputDown THEN
	GVL.EventLogger.print3(level:=TcEventSeverity.Warning, str1:='Both button pressed', str2:='', str3:=getSource());
	stopAll();
	pressedUpMiliseconds := 0;
	pressedDownMiliseconds := 0;
	justStopped := TRUE;
	JMP _stopped;
END_IF

manageConsecutiveClicks();

//moving any direction 
IF isClosing OR isOpening THEN
	IF pressedUp.Q OR pressedDown.Q THEN
		GVL.EventLogger.print3(level:=TcEventSeverity.Info, str1:='Button pressed during shutter move', str2:='', str3:=getSource());
				
		IF longDistanceUp.Q OR longDistanceDown.Q THEN
			GVL.EventLogger.print3(level:=TcEventSeverity.Verbose, str1:='Long move aborted', str2:='', str3:=getSource());
		END_IF
		stopAll();
		justStopped := TRUE;
		JMP _stopped;
	END_IF
END_IF

IF (releasedDown.Q OR releasedUp.Q) AND justStopped THEN
	justStopped := FALSE;
	GVL.EventLogger.print3(level:=TcEventSeverity.Verbose, str1:='Just stopped lock released', str2:='', str3:=getSource());
	JMP _stopped;
END_IF

goUpRequested := shortDistanceUp.Q OR longDistanceUp.Q;
goDownRequested := shortDistanceDown.Q OR longDistanceDown.Q;

IF goDownRequested AND NOT goUpRequested AND NOT isClosing THEN
	GVL.EventLogger.print3(level:=TcEventSeverity.Verbose, str1:='Go down requested', str2:='', str3:=getSource());
	moveDown();
	stopUp(preventMoving := TRUE);
ELSIF goUpRequested AND NOT goDownRequested AND NOT isOpening THEN
	GVL.EventLogger.print3(level:=TcEventSeverity.Verbose, str1:='Go up requested', str2:='', str3:=getSource());
	moveUp();
	stopDown(preventMoving := TRUE);
END_IF

//finished moving down
IF isClosing AND NOT goDownRequested AND NOT pressedDown.Q AND NOT manualControl THEN 
	GVL.EventLogger.print3(level:=TcEventSeverity.Verbose, str1:='Finished moving down', str2:='', str3:=getSource());
	stopDown(preventMoving := FALSE);
	requestedByGroupController := FALSE;
END_IF

//finished moving up
IF isOpening AND NOT goUpRequested AND NOT pressedUp.Q AND NOT manualControl THEN 
	GVL.EventLogger.print3(level:=TcEventSeverity.Verbose, str1:='Finished moving up', str2:='', str3:=getSource());
	stopUp(preventMoving := FALSE);
	requestedByGroupController := FALSE;
END_IF

IF requestedByGroupController THEN
	JMP _ret;	
END_IF

calculatePressedTimeMiliseconds();

IF releasedUp.Q THEN
	onReleasedUp();
END_IF

IF pressedUpMiliseconds >= 2000 THEN
	onContinuousHoldUp();
END_IF

IF releasedDown.Q THEN
	onReleasedDown();
END_IF

IF pressedDownMiliseconds >= 2000 THEN
	onContinuousHoldDown();
END_IF

_stopped :


_ret :
END_METHOD

METHOD PRIVATE manageConsecutiveClicks
VAR_INPUT
END_VAR

VAR

END_VAR
IF NOT inactivityTimeout.Q THEN
	consecutiveClicks := 0;
END_IF

IF pressedDown.Q THEN
	consecutiveClicks := consecutiveClicks + 1;
	inactivityTimeout(IN:= TRUE);
	GVL.EventLogger.print3(level:=TcEventSeverity.Verbose, str1:='consecutiveClicks=', str2:=TO_STRING(consecutiveClicks), str3:=getSource());
END_IF

IF consecutiveClicks >= 4 THEN
	consecutiveClicks := 0;
	doSpecialAction();
END_IF
END_METHOD

METHOD PRIVATE moveDown : BOOL
VAR_INPUT
END_VAR
IF canPrintGoDown THEN
	GVL.EventLogger.print3(level:=TcEventSeverity.Info, str1:='Roller shutter moving down', str2:='', str3:=getSource());
	canPrintGoDown := FALSE;
END_IF

//setOutputs(direction:=E_Direction.UP, state:=FALSE);
setOutputs(direction:=E_Direction.DOWN, state:=TRUE);
isClosing := TRUE;
END_METHOD

METHOD PUBLIC moveDownABit
VAR_INPUT
	requestedExternally : BOOL := FALSE;
END_VAR
GVL.EventLogger.print3(level:=TcEventSeverity.Info, str1:='Move down a bit', str2:= '', str3:=getSource());
//shortDistanceDown(IN:=releasedDown.Q);
shortDistanceDown(IN:=TRUE);
requestedByGroupController := requestedExternally;
END_METHOD

METHOD PUBLIC moveDownMax
VAR_INPUT
	requestedExternally : BOOL := FALSE;
END_VAR
GVL.EventLogger.print3(level:=TcEventSeverity.Info, str1:='Move down max', str2:= '', str3:=getSource());
longDistanceDown(IN:=TRUE);
requestedByGroupController := requestedExternally;
//longDistanceDown(IN:=releasedDown.Q);
GVL.EventLogger.print3(level:=TcEventSeverity.Verbose, str1:='Move requested externally?=', str2:= TO_STRING(requestedExternally), str3:=getSource());
END_METHOD

METHOD PRIVATE moveUp : BOOL
VAR_INPUT
END_VAR
IF canPrintGoUp THEN
	GVL.EventLogger.print3(level:=TcEventSeverity.Info, str1:='Roller shutter moving up', str2:='', str3:=getSource());
	canPrintGoUp := FALSE;
END_IF

//setOutputs(direction:=E_Direction.DOWN, state:=FALSE);
setOutputs(direction:=E_Direction.UP, state:=TRUE);
isOpening := TRUE;
END_METHOD

METHOD PUBLIC moveUpABit
VAR_INPUT
	requestedExternally : BOOL := FALSE;	
END_VAR
GVL.EventLogger.print3(level:=TcEventSeverity.Info, str1:='Move up a bit', str2:= '', str3:=getSource());
//shortDistanceUp(IN:=releasedUp.Q);
shortDistanceUp(IN:=TRUE);
requestedByGroupController := requestedExternally;
END_METHOD

METHOD PUBLIC moveUpMax
VAR_INPUT
	requestedExternally : BOOL := FALSE;
END_VAR
GVL.EventLogger.print3(level:=TcEventSeverity.Info, str1:='Move up max', str2:= '', str3:=getSource());
//longDistanceUp(IN:=releasedUp.Q);
longDistanceUp(IN:=TRUE);
requestedByGroupController := requestedExternally;
END_METHOD

METHOD onAnyPressedDown
VAR_INPUT
END_VAR
IF pressedDown.Q OR pressedUp.Q THEN
	IF pressedDown.Q THEN
		GVL.EventLogger.print3(level:=TcEventSeverity.Verbose, str1:='Button down pressed', str2:='', str3:=getSource());
	END_IF
	
	IF pressedUp.Q THEN
		GVL.EventLogger.print3(level:=TcEventSeverity.Verbose, str1:='Button up pressed', str2:='', str3:=getSource());
	END_IF
	
	requestedByGroupController := FALSE;
END_IF
END_METHOD

METHOD PRIVATE onContinuousHoldDown
VAR_INPUT
END_VAR
IF NOT manualControl THEN
	GVL.EventLogger.print3(level:=TcEventSeverity.Verbose, str1:='Start manual control by DOWN long press', str2:='', str3:=getSource());
END_IF

moveDown();
stopUp(preventMoving := TRUE);
manualControl := TRUE;
END_METHOD

METHOD PRIVATE onContinuousHoldUp
VAR_INPUT
END_VAR
IF NOT manualControl THEN
	GVL.EventLogger.print3(level:=TcEventSeverity.Verbose, str1:='Start manual control by UP long press', str2:='', str3:=getSource());
END_IF

moveUp();
stopDown(preventMoving := TRUE);
manualControl := TRUE;
END_METHOD

METHOD PRIVATE onReleasedDown : BOOL
VAR_INPUT
END_VAR
GVL.EventLogger.print3(level:=TcEventSeverity.Verbose, str1:='Button down released after ', str2:=TO_STRING(pressedDownMiliseconds), str3:=getSource());
manualControl := FALSE;
GVL.EventLogger.print3(level:=TcEventSeverity.Verbose, str1:='pressedDownMiliseconds=', str2:= TO_STRING(pressedDownMiliseconds), str3:=getSource());

IF pressedDownMiliseconds > 10 AND pressedDownMiliseconds < 500 THEN
	//move a bit down
	moveDownABit(requestedExternally:= FALSE);
ELSIF pressedDownMiliseconds >= 500 AND pressedDownMiliseconds < 2000 THEN
	//move max down
	moveDownMax(requestedExternally:= FALSE);
ELSIF pressedDownMiliseconds >= 2000 THEN
	//stop
	stopAll();
END_IF

pressedDownMiliseconds := 0;
END_METHOD

METHOD PRIVATE onReleasedUp : BOOL
VAR_INPUT
END_VAR
GVL.EventLogger.print3(level:=TcEventSeverity.Verbose, str1:='Button up released after ', str2:=TO_STRING(pressedUpMiliseconds), str3:=getSource());
manualControl := FALSE;
GVL.EventLogger.print3(level:=TcEventSeverity.Verbose, str1:='pressedUpMiliseconds=', str2:= TO_STRING(pressedUpMiliseconds), str3:=getSource());

IF pressedUpMiliseconds > 10 AND pressedUpMiliseconds < 500 THEN
	//move a bit up
	moveUpABit(requestedExternally:= FALSE);
ELSIF pressedUpMiliseconds >= 500 AND pressedUpMiliseconds < 2000 THEN
	//move max down
	moveUpMax(requestedExternally:= FALSE);
ELSIF pressedUpMiliseconds >= 2000 THEN
	//stop
	stopAll();
END_IF

pressedUpMiliseconds := 0;
END_METHOD

METHOD PRIVATE setOutputs
VAR_INPUT
	direction : E_Direction;
	state : BOOL;
END_VAR

VAR
	i : INT;
	state_as_text : STRING := 'abc';
END_VAR
IF manualControl THEN 
	JMP _bypass;
END_IF

state_as_text := TO_STRING(state);

CASE direction OF
	
	E_Direction.UP:
		GVL.EventLogger.print3(level:=TcEventSeverity.Info, str1:='set UP to: ', str2:= state_as_text, str3:=getSource());
		FOR i := 1 TO MAX_OUTPUTS_PER_LEVEL BY 1 DO
			up_outputs[i] := state;
		END_FOR
		
	E_Direction.DOWN:
		GVL.EventLogger.print3(level:=TcEventSeverity.Info, str1:='set DOWN to: ', str2:= state_as_text, str3:=getSource());	
		FOR i := 1 TO MAX_OUTPUTS_PER_LEVEL BY 1 DO
			down_outputs[i] := state;
		END_FOR
		
END_CASE

_bypass :
END_METHOD

METHOD stopAll : BOOL
VAR_INPUT
END_VAR
GVL.EventLogger.print3(level:=TcEventSeverity.Info, str1:='Stopping roller shutter', str2:='', str3:=getSource());
stopDown(preventMoving := FALSE);
stopUp(preventMoving := FALSE);
END_METHOD

METHOD stopDown : BOOL
VAR_INPUT
	preventMoving : BOOL := FALSE;
END_VAR
IF canPrintGoUp THEN
	IF preventMoving THEN
		GVL.EventLogger.print3(level:=TcEventSeverity.Verbose, str1:='Roller shutter moving down prevented', str2:='', str3:=getSource());
	ELSE
		GVL.EventLogger.print3(level:=TcEventSeverity.Info, str1:='Roller shutter moving down stopped', str2:='', str3:=getSource());
	END_IF
END_IF

canPrintGoDown := TRUE;
setOutputs(direction:=E_Direction.DOWN, state:=FALSE);
isClosing := FALSE;

stopDownTimers();
END_METHOD

METHOD stopDownTimers
VAR_INPUT
END_VAR
shortDistanceDown(PT := T#0S);
longDistanceDown(PT := T#0S);

shortDistanceDown(PT := shortTime);
longDistanceDown(PT := longTime);
END_METHOD

METHOD stopUp : BOOL
VAR_INPUT
	preventMoving : BOOL := FALSE;
END_VAR
IF canPrintGoDown THEN
	IF preventMoving THEN
		GVL.EventLogger.print3(level:=TcEventSeverity.Verbose, str1:='Roller shutter moving up prevented', str2:='', str3:=getSource());
	ELSE
		GVL.EventLogger.print3(level:=TcEventSeverity.Info, str1:='Roller shutter moving up stopped', str2:='', str3:=getSource());
	END_IF
END_IF


canPrintGoUp := TRUE;
setOutputs(direction:=E_Direction.UP, state:=FALSE);
isOpening:= FALSE;

stopUpTimers();
END_METHOD

METHOD stopUpTimers
VAR_INPUT
END_VAR
shortDistanceUp(PT := T#0S);
longDistanceUp(PT := T#0S);
shortDistanceUp(PT := shortTime);
longDistanceUp(PT := longTime);
END_METHOD

END_FUNCTION_BLOCK

// ---- POUs/log_persistence/EventLogger.TcPOU
FUNCTION_BLOCK EventLogger
VAR
	EventBuffer : ARRAY[1..EVENT_BUFFER_MAX_SIZE] OF ST_Event;
	CurrentEventBufferIndex : INT := 0;
	_PersistentEventStorage : I_PersistentEventStorage;
END_VAR
VAR CONSTANT
	EVENT_BUFFER_MAX_SIZE : INT := 100;
END_VAR

METHOD PUBLIC AddEvent : BOOL
VAR_INPUT
	eEventType : E_EventType;
	eEventSeverity : TcEventSeverity;
	nEventIdentity : UDINT;
	sEventText : STRING(255);
END_VAR
IF NOT IsEventBufferFull() THEN
	//todo
	CurrentEventBufferIndex := CurrentEventBufferIndex + 1;
	EventBuffer[CurrentEventBufferIndex].eEventType := eEventType;
	EventBuffer[CurrentEventBufferIndex].eEventSeverity := eEventSeverity;
	EventBuffer[CurrentEventBufferIndex].nEventIdentity := nEventIdentity;
	EventBuffer[CurrentEventBufferIndex].sEventText := sEventText;
	F_UpdateEventTimestampWithSystemTime(stEvent := EventBuffer[CurrentEventBufferIndex]); 
	AddEvent := TRUE;
ELSE
	AddEvent := FALSE;
END_IF

_PersistentEventStorage.StoreEvent(stEvent := EventBuffer[CurrentEventBufferIndex]);
END_METHOD

METHOD PUBLIC appendStrings : STRING(255)
VAR_INPUT
	str1 : STRING(255) := '';
	str2 : STRING(255) := '';
	str3 : STRING(255) := '';
END_VAR
VAR
	temp : STRING(255);
END_VAR
temp := CONCAT(STR1:=str1, STR2:=str2);
temp := CONCAT(STR1:=temp, STR2:=str3);
appendStrings := temp;
END_METHOD

METHOD FB_Init : BOOL
VAR_INPUT
	bInitRetains : BOOL;
	bInCopyCode : BOOL;
	iPersistentEventStorage : I_PersistentEventStorage;
END_VAR
_PersistentEventStorage := iPersistentEventStorage;
END_METHOD

METHOD PRIVATE IsEventBufferFull : BOOL
IF (CurrentEventBufferIndex + 1) >= EVENT_BUFFER_MAX_SIZE THEN
	IsEventBufferFull := TRUE;
ELSE
	IsEventBufferFull := FALSE;
END_IF
END_METHOD

METHOD print1 : BOOL
VAR_INPUT
	level : TcEventSeverity;
	str1 : STRING;
END_VAR

VAR
	enum_as_text : STRING;
END_VAR
CASE level OF
	TcEventSeverity.Critical:
		enum_as_text := '[CRITICAL] ';
	TcEventSeverity.Error:
		enum_as_text := '[ERROR] ';
	TcEventSeverity.Warning:
		enum_as_text := '[WARNING] ';		
	TcEventSeverity.Info:
		enum_as_text := '        [INFO] ';
	TcEventSeverity.Verbose:
		enum_as_text := '                        [VERBOSE] ';
END_CASE

IF (TO_SINT(level) >= MAIN.minimumLogSeverity) THEN
	ADSLOGSTR(ADSLOG_MSGTYPE_ERROR, 
              CONCAT(enum_as_text, str1), 
              '');
END_IF
END_METHOD

METHOD print2 : BOOL
VAR_INPUT
	level : TcEventSeverity;
	str1 : STRING;
	str2 : STRING;
END_VAR

VAR
	enum_as_text : STRING;
END_VAR
CASE level OF
	TcEventSeverity.Critical:
		enum_as_text := '[CRITICAL] ';
	TcEventSeverity.Error:
		enum_as_text := '[ERROR] ';
	TcEventSeverity.Warning:
		enum_as_text := '[WARNING] ';		
	TcEventSeverity.Info:
		enum_as_text := '        [INFO] ';
	TcEventSeverity.Verbose:
		enum_as_text := '                        [VERBOSE] ';
END_CASE

IF (TO_SINT(level) >= MAIN.minimumLogSeverity) THEN
	ADSLOGSTR(ADSLOG_MSGTYPE_ERROR, 
			  CONCAT(enum_as_text, str1), 
			  str2);
END_IF
END_METHOD

METHOD print3 : BOOL
VAR_INPUT
	level : TcEventSeverity;
	str1 : STRING(255);
	str2 : STRING(255);
	str3 : STRING(255);
END_VAR

VAR
	enum_as_text : STRING(255);
	val : STRING(255);
END_VAR
CASE level OF
	TcEventSeverity.Critical:
		enum_as_text := '[CRITICAL] ';
	TcEventSeverity.Error:
		enum_as_text := '[ERROR] ';
	TcEventSeverity.Warning:
		enum_as_text := '[WARNING] ';		
	TcEventSeverity.Info:
		enum_as_text := '[INFO] ';
	TcEventSeverity.Verbose:
		enum_as_text := '     [VERBOSE] ';
END_CASE

val := appendStrings(str1:= str1, str2:= str2, str3:= str3);

IF (TO_SINT(level) >= MAIN.minimumLogSeverity) THEN
	ADSLOGSTR(ADSLOG_MSGTYPE_ERROR, 
			  CONCAT(enum_as_text, val), 
			  '');
END_IF
END_METHOD

END_FUNCTION_BLOCK

// ---- POUs/log_persistence/F_UpdateEventTimestampWithSystemTime.TcPOU
FUNCTION F_UpdateEventTimestampWithSystemTime
VAR_INPUT
	stEvent : REFERENCE TO ST_Event;
END_VAR
VAR
	fbGETSYSTEMTIME : GETSYSTEMTIME;
	stFileTime : T_FILETIME;
END_VAR

fbGETSYSTEMTIME(timeLoDW => stFileTime.dwLowDateTime,
				timeHiDW => stFileTime.dwHighDateTime);
stEvent.dtTimestamp := FILETIME_TO_DT(fileTime := stFileTime);

END_FUNCTION

// ---- POUs/SequentialLightSwitch.TcPOU
FUNCTION_BLOCK SequentialLightSwitch

VAR CONSTANT
	MAX_OUTPUTS_PER_LEVEL : INT := GVL.MAX_LIGHT_OUTPUTS_PER_LEVEL;
END_VAR

VAR_INPUT
	ID : INT;
	name : STRING := 'Light switch';
	digitalInput : REFERENCE TO BOOL;
	
	small_outputs : REFERENCE TO ARRAY[1..MAX_OUTPUTS_PER_LEVEL] OF BOOL;
	medium_outputs : REFERENCE TO ARRAY[1..MAX_OUTPUTS_PER_LEVEL] OF BOOL;
	big_outputs : REFERENCE TO ARRAY[1..MAX_OUTPUTS_PER_LEVEL] OF BOOL;
	superstrong_outputs : REFERENCE TO ARRAY[1..MAX_OUTPUTS_PER_LEVEL] OF BOOL;
	
	levelsManaged : INT := 3; //max 4
	
	defaultDayOutput : E_OutputLevel;
	defaultNightOutput : E_OutputLevel;
END_VAR

VAR	
	initialized : BOOL := FALSE;
	isOn : BOOL := FALSE;
	smallOutputsSet : BOOL := FALSE;
	mediumOutputsSet : BOOL := FALSE;
	bigOutputsSet: BOOL := FALSE;
	superStrongOutputsSet: BOOL := FALSE;
	
	wasRecentlyActive : BOOL := FALSE;
	pressed : R_TRIG;
	released : F_TRIG;
	smallOutputTimer : TON := (PT := T#1S);
	mediumOutputTimer : TON := (PT := T#2S); 
	bigOutputTimer : TON := (PT := T#3S); 
	superStrongOutputTimer : TON := (PT := T#4S);
	inactivityTimeout : TP := (PT := T#1100MS);
	pressedTimer : TON := (PT := T#10S);
	pressedTimeMiliseconds : INT := 0;
	firstLongPress : BOOL := FALSE;
	turnedOnLongSelector : BOOL := FALSE;
	
	consecutiveClicks : INT := 0;
END_VAR

IF NOT initialized THEN
	initialized := TRUE;	
END_IF

METHOD doSpecialAction : BOOL
VAR_INPUT
END_VAR

VAR
	i: INT;
	groupController : GroupController;
END_VAR
CASE ID OF
		//TODO pamietac
	12:
		GVL.EventLogger.print3(level:=TcEventSeverity.Info, str1:='Special action for button 1 - ', str2:='turning off all lights', str3:=getSource());
		MAIN.groupController.requestLightsOff();
		
	17:
		GVL.EventLogger.print3(level:=TcEventSeverity.Info, str1:='Special action for button 2 - ', str2:='turning on all lights', str3:=getSource());
		MAIN.groupController.requestLightsOnDefault();
		
//	3:
//		GVL.EventLogger.print3(level:=TcEventSeverity.Info, str1:='Special action for button 3 - ', str2:='closing all shutters', str3:=getSource());
//		MAIN.groupController.requestShuttersClose();
		
END_CASE
END_METHOD

METHOD PRIVATE getSource : STRING(255)
VAR_INPUT
END_VAR

VAR
	details : STRING(255);
END_VAR
details := CONCAT(STR1:=' - light switch, ID: ', STR2:=TO_STRING(ID));
details := CONCAT(STR1:=details, STR2:=', digital input: ');
details := CONCAT(STR1:=details, STR2:=TO_STRING(digitalInput));
details := CONCAT(STR1:=details, STR2:=', name: ');
details := CONCAT(STR1:=details, STR2:=name);

getSource := details;
END_METHOD

METHOD PRIVATE inputsOutputsLoop
VAR_INPUT
END_VAR
pressed(CLK:= digitalInput);
released(CLK:= digitalInput);
smallOutputTimer(IN := digitalInput);
mediumOutputTimer(IN := digitalInput);
bigOutputTimer(IN := digitalInput);
superStrongOutputTimer(IN := digitalInput);
inactivityTimeout(IN := digitalInput);
pressedTimer(IN := digitalInput);
turnedOnLongSelector := isTurnedOnLongSelector();
END_METHOD

METHOD PRIVATE isTurnedOnLongSelector : BOOL
VAR_INPUT
END_VAR
isTurnedOnLongSelector := smallOutputsSet OR mediumOutputsSet OR bigOutputsSet OR superStrongOutputsSet;
END_METHOD

METHOD loop
VAR_INPUT
END_VAR

VAR
	number : DINT;
	boool : BOOL;
	str3: INT;
END_VAR
verifyIsTurnedOn();
inputsOutputsLoop();


IF NOT inactivityTimeout.Q THEN
	firstLongPress := FALSE;	
END_IF

IF digitalInput THEN
	IF TIME_TO_INT(pressedTimer.ET) <> 0 THEN
		pressedTimeMiliseconds := TIME_TO_INT(pressedTimer.ET);
	END_IF
END_IF

IF wasRecentlyActive AND NOT digitalInput AND NOT inactivityTimeout.Q THEN	
	GVL.EventLogger.print3(level:= TcEventSeverity.Verbose, str1:='Activity timeout', str2:= '', str3:=getSource());
	consecutiveClicks := 0;
	wasRecentlyActive := FALSE;
END_IF

IF pressed.Q THEN
	GVL.EventLogger.print3(level:=TcEventSeverity.Info, str1:='Button pressed', str2:= '', str3:=getSource());
	consecutiveClicks := consecutiveClicks + 1;
	GVL.EventLogger.print3(level:=TcEventSeverity.Verbose, str1:='consecutiveClicks=', str2:= TO_STRING(consecutiveClicks), str3:=getSource());
	GVL.EventLogger.print3(level:=TcEventSeverity.Verbose, str1:='isOn=', str2:= TO_STRING(isOn), str3:=getSource());
	GVL.EventLogger.print3(level:=TcEventSeverity.Verbose, str1:='firstLongPress=', str2:= TO_STRING(firstLongPress), str3:=getSource());
	
END_IF

IF released.Q THEN
	GVL.EventLogger.print3(level:=TcEventSeverity.Info, str1:='Released after ', str2:= TO_STRING(pressedTimeMiliseconds), str3:=getSource());
	GVL.EventLogger.print3(level:=TcEventSeverity.Verbose, str1:='isOn=', str2:= TO_STRING(isOn), str3:=getSource());
	GVL.EventLogger.print3(level:=TcEventSeverity.Verbose, str1:='turnedOnLongSelector=', str2:= TO_STRING(turnedOnLongSelector), str3:=getSource());
	GVL.EventLogger.print3(level:=TcEventSeverity.Verbose, str1:='firstLongPress=', str2:= TO_STRING(firstLongPress), str3:=getSource());	
	IF isON AND NOT turnedOnLongSelector AND NOT firstLongPress THEN
		GVL.EventLogger.print3(level:=TcEventSeverity.Info, str1:='Lights turned off', str2:= '', str3:=getSource());
		turnOff();
	ELSE		
		GVL.EventLogger.print3(level:=TcEventSeverity.Verbose, str1:='wasRecentlyActive=', str2:= TO_STRING(wasRecentlyActive), str3:=getSource());
		IF pressedTimeMiliseconds >= 0 AND pressedTimeMiliseconds <= 300  THEN
			GVL.EventLogger.print3(level:=TcEventSeverity.Verbose, str1:='Quick press released after ', str2:= TO_STRING(pressedTimeMiliseconds), str3:=getSource());
			GVL.EventLogger.print3(level:=TcEventSeverity.Verbose, str1:='firstLongPress=', str2:= TO_STRING(firstLongPress), str3:=getSource());
			IF NOT firstLongPress THEN
				turnOnDefault();
			END_IF
		ELSE 
			IF pressedTimeMiliseconds > 300 AND pressedTimeMiliseconds < 1000 THEN
				GVL.EventLogger.print3(level:=TcEventSeverity.Verbose, str1:='Long press released after ', str2:= TO_STRING(pressedTimeMiliseconds), str3:=getSource());
				GVL.EventLogger.print3(level:=TcEventSeverity.Verbose, str1:='Turn ON strongest as long press', str2:= '', str3:=getSource());
				turnOnStrongestOutput();
			END_IF 
		END_IF
	END_IF
	
	wasRecentlyActive := TRUE;
	pressedTimeMiliseconds := TIME_TO_INT(pressedTimer.ET);
END_IF

IF consecutiveClicks >= 3 THEN
	consecutiveClicks := 0;
	doSpecialAction();
END_IF

manageLongPress();
END_METHOD

METHOD PRIVATE manageLongPress
VAR_INPUT
END_VAR
IF levelsManaged >= 1 AND TIME_TO_DWORD(pressedTimer.ET) >= 1000 THEN
	IF NOT smallOutputsSet THEN
		setOutputs(outputLevel := E_OutputLevel.SMALL, state := TRUE);
		GVL.EventLogger.print3(level:=TcEventSeverity.Verbose, str1:='Long press turn on output ', str2:=TO_STRING(E_OutputLevel.SMALL), str3:=getSource());
	END_IF
END_IF

IF levelsManaged >= 2 AND TIME_TO_DWORD(pressedTimer.ET) >= 2000 THEN
	IF NOT mediumOutputsSet THEN
		setOutputs(outputLevel := E_OutputLevel.MEDIUM, state := TRUE);
		GVL.EventLogger.print3(level:=TcEventSeverity.Verbose, str1:='Long press turn on output', str2:=TO_STRING(E_OutputLevel.SMALL), str3:=getSource());
	END_IF
END_IF

IF levelsManaged >= 3 AND TIME_TO_DWORD(pressedTimer.ET) >= 3000 THEN
	IF NOT bigOutputsSet THEN
		setOutputs(outputLevel := E_OutputLevel.BIG, state := TRUE);
		GVL.EventLogger.print3(level:=TcEventSeverity.Verbose, str1:='Long press turn on output', str2:=TO_STRING(E_OutputLevel.SMALL), str3:=getSource());
	END_IF
END_IF

IF levelsManaged >= 4 AND TIME_TO_DWORD(pressedTimer.ET) >= 4000 THEN
	IF NOT superStrongOutputsSet THEN
		setOutputs(outputLevel := E_OutputLevel.SUPERSTRONG, state := TRUE);
		GVL.EventLogger.print3(level:=TcEventSeverity.Verbose, str1:='Long press turn on output', str2:=TO_STRING(E_OutputLevel.SMALL), str3:=getSource());
	END_IF
END_IF
END_METHOD

METHOD PRIVATE setOutputs
VAR_INPUT
	outputLevel : E_OutputLevel;
	state : BOOL;
END_VAR

VAR
	i : INT;
	state_as_text : STRING := 'abc';
END_VAR
state_as_text := TO_STRING(state);

CASE outputLevel OF
	
	E_OutputLevel.SMALL:
		GVL.EventLogger.print3(level:=TcEventSeverity.Info, str1:='Set SMALL outputs to: ', str2:= state_as_text, str3:=getSource());
		FOR i := 1 TO MAX_OUTPUTS_PER_LEVEL BY 1 DO
			small_outputs[i] := state;
		END_FOR
		
	E_OutputLevel.MEDIUM:
		GVL.EventLogger.print3(level:=TcEventSeverity.Info, str1:='Set MEDIUM outputs to: ', str2:= state_as_text, str3:=getSource());	
		FOR i := 1 TO MAX_OUTPUTS_PER_LEVEL BY 1 DO
			medium_outputs[i] := state;
		END_FOR
		
	E_OutputLevel.BIG:
		GVL.EventLogger.print3(level:=TcEventSeverity.Info, str1:='Set BIG outputs to: ', str2:= state_as_text, str3:=getSource());
		FOR i := 1 TO MAX_OUTPUTS_PER_LEVEL BY 1 DO
			big_outputs[i] := state;
		END_FOR
		
	E_OutputLevel.SUPERSTRONG:
		GVL.EventLogger.print3(level:=TcEventSeverity.Info, str1:='Set SUPERSTRONG outputs to: ', str2:= state_as_text, str3:=getSource());
		FOR i := 1 TO MAX_OUTPUTS_PER_LEVEL BY 1 DO
			superstrong_outputs[i] := state;
		END_FOR
		
END_CASE
END_METHOD

METHOD PUBLIC turnOff
VAR_INPUT
END_VAR

VAR 
	i : INT;
END_VAR
CASE levelsManaged OF
	1 :
		FOR i := 1 TO MAX_OUTPUTS_PER_LEVEL BY 1 DO
			small_outputs[i] := FALSE;
		END_FOR

	2 :
		FOR i := 1 TO MAX_OUTPUTS_PER_LEVEL BY 1 DO
			small_outputs[i] := FALSE;
			medium_outputs[i] := FALSE;
		END_FOR
	
	3 :
		FOR i := 1 TO MAX_OUTPUTS_PER_LEVEL BY 1 DO
			small_outputs[i] := FALSE;
			medium_outputs[i] := FALSE;
			big_outputs[i] := FALSE;
		END_FOR
		
	4 :
		FOR i := 1 TO MAX_OUTPUTS_PER_LEVEL BY 1 DO
			small_outputs[i] := FALSE;
			medium_outputs[i] := FALSE;
			big_outputs[i] := FALSE;
			superstrong_outputs[i] := FALSE;
		END_FOR

END_CASE

isOn := FALSE;
END_METHOD

METHOD PUBLIC turnOnDefault
VAR_INPUT
END_VAR
IF MAIN.isDay THEN
	GVL.EventLogger.print3(level:=TcEventSeverity.Verbose, str1:='turn ON default for daytime: ', str2:= TO_STRING(defaultDayOutput), str3:=getSource());
	setOutputs(outputLevel := defaultDayOutput, state := TRUE);
ELSE
	GVL.EventLogger.print3(level:=TcEventSeverity.Verbose, str1:='turn ON default for nighttime: ', str2:= TO_STRING(defaultNightOutput), str3:=getSource());
	setOutputs(outputLevel := defaultNightOutput, state := TRUE);
END_IF

isOn := TRUE;
END_METHOD

METHOD turnOnStrongestOutput
VAR_INPUT
END_VAR

VAR
	i : INT;
END_VAR
CASE levelsManaged OF
	1:
		setOutputs(outputLevel := E_OutputLevel.SMALL, state := TRUE);
		setOutputs(outputLevel := E_OutputLevel.MEDIUM, state := FALSE);
		setOutputs(outputLevel := E_OutputLevel.BIG, state := FALSE);
		setOutputs(outputLevel := E_OutputLevel.SUPERSTRONG, state := FALSE);
	2:
		setOutputs(outputLevel := E_OutputLevel.SMALL, state := FALSE);
		setOutputs(outputLevel := E_OutputLevel.MEDIUM, state := TRUE);
		setOutputs(outputLevel := E_OutputLevel.BIG, state := FALSE);
		setOutputs(outputLevel := E_OutputLevel.SUPERSTRONG, state := FALSE);
		
	3:
		setOutputs(outputLevel := E_OutputLevel.SMALL, state := FALSE);
		setOutputs(outputLevel := E_OutputLevel.MEDIUM, state := FALSE);
		setOutputs(outputLevel := E_OutputLevel.BIG, state := TRUE);
		setOutputs(outputLevel := E_OutputLevel.SUPERSTRONG, state := FALSE);
		
	4:
		setOutputs(outputLevel := E_OutputLevel.SMALL, state := FALSE);
		setOutputs(outputLevel := E_OutputLevel.MEDIUM, state := FALSE);
		setOutputs(outputLevel := E_OutputLevel.BIG, state := FALSE);
		setOutputs(outputLevel := E_OutputLevel.SUPERSTRONG, state := TRUE);
		
END_CASE

isOn := TRUE;
END_METHOD

METHOD PRIVATE verifyIsTurnedOn
VAR_INPUT
END_VAR

VAR
	i : INT;
END_VAR
isOn := FALSE;
smallOutputsSet := FALSE;
mediumOutputsSet := FALSE;
bigOutputsSet := FALSE;
superStrongOutputsSet := FALSE;

IF levelsManaged >= 1 THEN
	FOR i := 1 TO MAX_OUTPUTS_PER_LEVEL BY 1 DO
		IF small_outputs[i] = TRUE THEN
			isOn := TRUE;
			smallOutputsSet := TRUE;
		END_IF
	END_FOR
END_IF

IF levelsManaged >= 2 THEN
	FOR i := 1 TO MAX_OUTPUTS_PER_LEVEL BY 1 DO
		IF medium_outputs[i] = TRUE THEN
			isOn := TRUE;
			mediumOutputsSet := TRUE;
		END_IF
	END_FOR
END_IF

IF levelsManaged >= 3 THEN
	FOR i := 1 TO MAX_OUTPUTS_PER_LEVEL BY 1 DO
		IF big_outputs[i] = TRUE THEN
			isOn := TRUE;
			bigOutputsSet := TRUE;
		END_IF
	END_FOR
END_IF

IF levelsManaged >= 4 THEN
	FOR i := 1 TO MAX_OUTPUTS_PER_LEVEL BY 1 DO
		IF superstrong_outputs[i] = TRUE THEN
			isOn := TRUE;
			superStrongOutputsSet := TRUE;
		END_IF
	END_FOR
END_IF


RETURN;
END_METHOD

END_FUNCTION_BLOCK

// ---- POUs/SimpleButton.TcPOU
FUNCTION_BLOCK SimpleButton

VAR CONSTANT
	MAX_OUTPUTS : INT := GVL.MAX_SIMPLE_OUTPUTS;
END_VAR

VAR_INPUT
	ID : INT;
	name : STRING := 'Simple button';
	digitalInput : REFERENCE TO BOOL;
	outputs : REFERENCE TO ARRAY[1..MAX_OUTPUTS] OF BOOL;
	runAsYouPress : BOOL := FALSE;
	holdTime : TIME := T#10MS;
    withHold : BOOL := FALSE;
	lightSwitch : BOOL := FALSE;
END_VAR

VAR_OUTPUT
END_VAR

VAR
	isOn : BOOL := FALSE;
	printed : BOOL := FALSE;
	pressed : R_TRIG;
	released : F_TRIG;
	holdTimer : TP := (PT := holdTime);
	readyToBeTurnedOff : BOOL := FALSE;
	inactivityTimeout : TP := (PT := T#1100MS);
	consecutiveClicks : INT := 0;
END_VAR

holdTimer(PT:= holdTime);

METHOD doSpecialAction : BOOL
VAR_INPUT
END_VAR

VAR
	i: INT;
END_VAR
CASE ID OF
	//TODO pamietac
	33:
		GVL.EventLogger.print3(level:=TcEventSeverity.Info, str1:='Special action for button 1 - ', str2:='turning off all lights', str3:=getSource());
		MAIN.groupController.requestLightsOff();
		
	2:
		GVL.EventLogger.print3(level:=TcEventSeverity.Info, str1:='Special action for button 2 - ', str2:='opening on all lights', str3:=getSource());
		MAIN.groupController.requestLightsOnDefault();
		
//	1:
	//	GVL.EventLogger.print3(level:=TcEventSeverity.Info, str1:='Special action for button 3 - ', str2:='closing all shutters', str3:=getSource());
		//MAIN.groupController.requestShuttersClose();
		
END_CASE
END_METHOD

METHOD PRIVATE getSource : STRING
VAR_INPUT
END_VAR

VAR
	details : STRING;
END_VAR
details := CONCAT(STR1:=' - simple button, ID: ', STR2:=TO_STRING(ID));
details := CONCAT(STR1:=details, STR2:=', digital input: ');
details := CONCAT(STR1:=details, STR2:=TO_STRING(digitalInput));
details := CONCAT(STR1:=details, STR2:=', name: ');
details := CONCAT(STR1:=details, STR2:=name);

getSource := details;
END_METHOD

METHOD PRIVATE inputsOutputsLoop
VAR_INPUT
END_VAR
pressed(CLK:= digitalInput);
released(CLK:= digitalInput);
holdTimer(IN:= FALSE);
inactivityTimeout(IN:= FALSE);
END_METHOD

METHOD PUBLIC isLightSwitch : BOOL
VAR_INPUT
END_VAR
isLightSwitch := lightSwitch;
END_METHOD

METHOD PUBLIC loop : BOOL
VAR_INPUT
END_VAR
verifyIsTurnedOn();
inputsOutputsLoop();

IF pressed.Q THEN
	GVL.EventLogger.print3(level:= TcEventSeverity.Info, str1:='Button pressed', str2:= '', str3:=getSource());
	printed := FALSE;
END_IF

IF released.Q THEN
	GVL.EventLogger.print3(level:= TcEventSeverity.Info, str1:='Button released', str2:= '', str3:=getSource());
	printed := FALSE;
END_IF

manageConsecutiveClicks();

IF runAsYouPress THEN
	setOutputs(state:= digitalInput);
ELSE
	IF pressed.Q THEN
		IF isOn THEN 			//turned on -> lets turn off
			turnOff();
			stopHoldTimer();
		ELSE 					//turned off -> lets turn on
			turnOn();
			IF withHold THEN
				GVL.EventLogger.print3(level:= TcEventSeverity.Verbose, str1:='Button turned ON with hold time miliseconds=', str2:=TO_STRING(TIME_TO_INT(holdTime)), str3:=getSource());
				holdTimer(IN:= TRUE);
				readyToBeTurnedOff := TRUE;
			END_IF
		END_IF
	END_IF
	
	IF withHold AND readyToBeTurnedOff AND NOT holdTimer.Q THEN
		turnOff();
		readyToBeTurnedOff := FALSE;
		GVL.EventLogger.print3(level:= TcEventSeverity.Verbose, str1:='Button turned OFF automatically after hold time miliseconds=', str2:=TO_STRING(TIME_TO_INT(holdTime)), str3:=getSource());
	END_IF
END_IF
END_METHOD

METHOD PRIVATE manageConsecutiveClicks
VAR_INPUT
END_VAR

VAR

END_VAR
IF NOT inactivityTimeout.Q THEN
	consecutiveClicks := 0;
END_IF

IF pressed.Q THEN
	consecutiveClicks := consecutiveClicks + 1;
	inactivityTimeout(IN:= TRUE);
	GVL.EventLogger.print3(level:=TcEventSeverity.Verbose, str1:='consecutiveClicks=', str2:=TO_STRING(consecutiveClicks), str3:=getSource());
END_IF

IF consecutiveClicks >= 3 THEN
	consecutiveClicks := 0;
	doSpecialAction();
END_IF
END_METHOD

METHOD setOutputs
VAR_INPUT
	state : BOOL;
END_VAR

VAR
	i : INT;
	state_as_text : STRING := 'abc';
END_VAR
state_as_text := TO_STRING(state);

IF NOT printed THEN
	GVL.EventLogger.print3(level:=TcEventSeverity.Info, str1:='Set outputs to: ', str2:= state_as_text, str3:=getSource());
	printed := TRUE;
END_IF

FOR i := 1 TO MAX_OUTPUTS BY 1 DO
	outputs[i] := state;
END_FOR
END_METHOD

METHOD stopHoldTimer
VAR_INPUT
END_VAR
holdTimer(PT:=T#0S);
holdTimer(PT:=holdTime);
END_METHOD

METHOD PUBLIC turnOff
VAR_INPUT
END_VAR
setOutputs(state:= FALSE);
END_METHOD

METHOD PUBLIC turnOn
VAR_INPUT
END_VAR
setOutputs(state:= TRUE);
END_METHOD

METHOD PRIVATE verifyIsTurnedOn
VAR_INPUT
END_VAR

VAR
	i : INT;
END_VAR
isOn := FALSE;
FOR i := 1 TO MAX_OUTPUTS BY 1 DO
	IF outputs[i] = TRUE THEN
		isOn := TRUE;
		RETURN;
	END_IF
END_FOR

RETURN;
END_METHOD

END_FUNCTION_BLOCK

// ---- POUs/UpStopDownButton.TcPOU
FUNCTION_BLOCK UpStopDownButton

VAR CONSTANT
	MAX_OUTPUTS_PER_LEVEL : INT := 3;
END_VAR

VAR_INPUT
	ID : INT;
	name : STRING := 'UpStopDown button';
	digitalInput : REFERENCE TO BOOL;
	outputs : REFERENCE TO ARRAY[1..MAX_OUTPUTS_PER_LEVEL] OF BOOL;
	defaultFirstClickDirection : E_Direction;
END_VAR
VAR_OUTPUT
END_VAR
VAR
	pressed : R_TRIG;
	state : E_Direction := E_Direction.STOP;
    previousState : E_Direction := E_Direction.STOP;
	returnTimer : TP := (PT := T#500MS);
	
	readyToRelease : BOOL := FALSE;
END_VAR

METHOD getSource : STRING
VAR_INPUT
END_VAR

VAR
	details : STRING;
END_VAR
details := CONCAT(STR1:=' - up-stop-down button, ID: ', STR2:=TO_STRING(ID));
details := CONCAT(STR1:=details, STR2:=', digital input: ');
details := CONCAT(STR1:=details, STR2:=TO_STRING(digitalInput));
details := CONCAT(STR1:=details, STR2:=', name: ');
details := CONCAT(STR1:=details, STR2:=name);

getSource := details;
END_METHOD

METHOD loop : BOOL
VAR_INPUT
END_VAR
pressed(CLK:= digitalInput);
returnTimer(IN:= pressed.Q);

IF pressed.Q THEN
	readyToRelease := TRUE;
	
	GVL.EventLogger.print3(level:= TcEventSeverity.Verbose, str1:='Just before pressing Previous state=', str2:= TO_STRING(previousState), str3:=getSource());
	GVL.EventLogger.print3(level:= TcEventSeverity.Verbose, str1:='Just before pressing Current state=', str2:=TO_STRING(state), str3:=getSource());
	GVL.EventLogger.print3(level:= TcEventSeverity.Info, str1:='Pressed button=', str2:='', str3:=getSource());
	
	manageStatesAfterPressed();
	
	GVL.EventLogger.print3(level:= TcEventSeverity.Verbose, str1:='After pressing Previous state=', str2:= TO_STRING(previousState), str3:=getSource());
	GVL.EventLogger.print3(level:= TcEventSeverity.Verbose, str1:='After pressing Current state=', str2:=TO_STRING(state), str3:=getSource());

	setOutputs(state:= TRUE);

END_IF

IF NOT returnTimer.Q AND readyToRelease THEN
	setOutputs(state:= FALSE);
	readyToRelease := FALSE;
END_IF
END_METHOD

METHOD manageStatesAfterPressed
VAR_INPUT
END_VAR
CASE state OF
	E_Direction.STOP:
		CASE previousState OF
			E_Direction.STOP:
				state := defaultFirstClickDirection;
			E_Direction.DOWN:
				state := E_Direction.UP;
			E_Direction.UP:
				state := E_Direction.DOWN;
		END_CASE
		previousState := E_Direction.STOP;
		
	E_Direction.DOWN:
		state := E_Direction.STOP;
		previousState := E_Direction.DOWN;
		
	E_Direction.UP:
		state := E_Direction.STOP;
		previousState := E_Direction.UP;
END_CASE
END_METHOD

METHOD setOutputs
VAR_INPUT
	state : BOOL;
END_VAR

VAR
	i : INT;
	state_as_text : STRING := 'abc';
END_VAR
state_as_text := TO_STRING(state);

GVL.EventLogger.print3(level:=TcEventSeverity.Info, str1:='Set outputs to: ', str2:= state_as_text, str3:=getSource());
FOR i := 1 TO MAX_OUTPUTS_PER_LEVEL BY 1 DO
	outputs[i] := state;
END_FOR
END_METHOD

END_FUNCTION_BLOCK

// ---- POUs/log_persistence/FB_CsvPersistentEventStorage.TcPOU
FUNCTION_BLOCK FB_CsvPersistentEventStorage IMPLEMENTS I_PersistentEventStorage
VAR_INPUT
	fbFileOpen : FB_FileOpen := (sPathName := 'C:\Events.log', nMode := FOPEN_MODEAPPEND OR FOPEN_MODETEXT);
	fbFilePuts : FB_FilePuts;
	fbFileClose : FB_FileClose;
	eWriteState : (FILE_OPEN_TRIGGER, FILE_OPEN, WAIT_FOR_EVENT, WRITE_EVENT_TRIGGER, WRITE_EVENT, FILE_CLOSE_TRIGGER, FILE_CLOSE, ERROR);
	stEventWrittenToFile : ST_Event;
	CsvString : T_MaxString;
	FILE_CLOSE_TRIGGER : INT;
END_VAR
VAR_OUTPUT
END_VAR
VAR
	FILE_CLOSE: INT;
END_VAR

CASE eWriteState OF
	FILE_OPEN_TRIGGER:
		fbFileOpen(bExecute := TRUE);
		eWriteState := FILE_OPEN;
	
	FILE_OPEN:
		fbFileOpen(bExecute := FALSE);
		IF fbFileOpen.bError THEN
			eWriteSTate := ERROR;
		ELSIF NOT fbFileOpen.bBusy AND fbFileOpen.hFile <> 0 THEN
			eWriteState := WAIT_FOR_EVENT;
		END_IF
		
	WAIT_FOR_EVENT:
		//do nothing
		
	WRITE_EVENT_TRIGGER:
		CsvString := CreateCsvString(stEvent := stEventWrittenToFile);
		fbFilePuts(bExecute := TRUE,
					sLine := CsvString,
					hFile := fbFileOpen.hFile);
			
	FILE_CLOSE_TRIGGER:
		fbFileClose(bExecute := TRUE,
					hFile := fbFileOpen.hFile);
		eWriteState := FILE_CLOSE;
		
	FILE_CLOSE:
		fbFileClose(bExecute := FALSE);
		IF fbFileClose.bError THEN
			eWriteState := ERROR;
		ELSIF NOT fbFileClose.bBusy THEN
			eWriteState := FILE_OPEN_TRIGGER;
		END_IF
		
	ERROR:
		//DO NOTHING
END_CASE

METHOD CreateCsvString : T_MaxString
VAR_INPUT
	stEvent : REFERENCE TO ST_Event;
END_VAR
VAR
	TempString : T_MaxString;
END_VAR
TempString := TO_STRING(stEvent.eEventType);
TempString := CONCAT(STR1 := TempString, STR2 := ',');
TempString := CONCAT(STR1 := TempString, STR2 := TO_STRING(stEvent.eEventSeverity));
TempString := CONCAT(STR1 := TempString, STR2 := ',');
TempString := CONCAT(STR1 := TempString, STR2 := TO_STRING(stEvent.nEventIdentity));
TempString := CONCAT(STR1 := TempString, STR2 := ',');
TempString := CONCAT(STR1 := TempString, STR2 := stEvent.sEventText);
TempString := CONCAT(STR1 := TempString, STR2 := ',');
TempString := CONCAT(STR1 := TempString, STR2 := TO_STRING(stEvent.dtTimestamp));
TempString := CONCAT(STR1 := TempString, STR2 := '$n');

CreateCsvString := TempString;
END_METHOD

METHOD StoreEvent
VAR_INPUT
	stEvent	: ST_Event;
END_VAR
IF eWriteState = WAIT_FOR_EVENT THEN
	eWriteState := WRITE_EVENT_TRIGGER;
	stEventWrittenToFile := stEvent;
END_IF
END_METHOD

END_FUNCTION_BLOCK

// ---- VISUs/Screen1.TcVIS
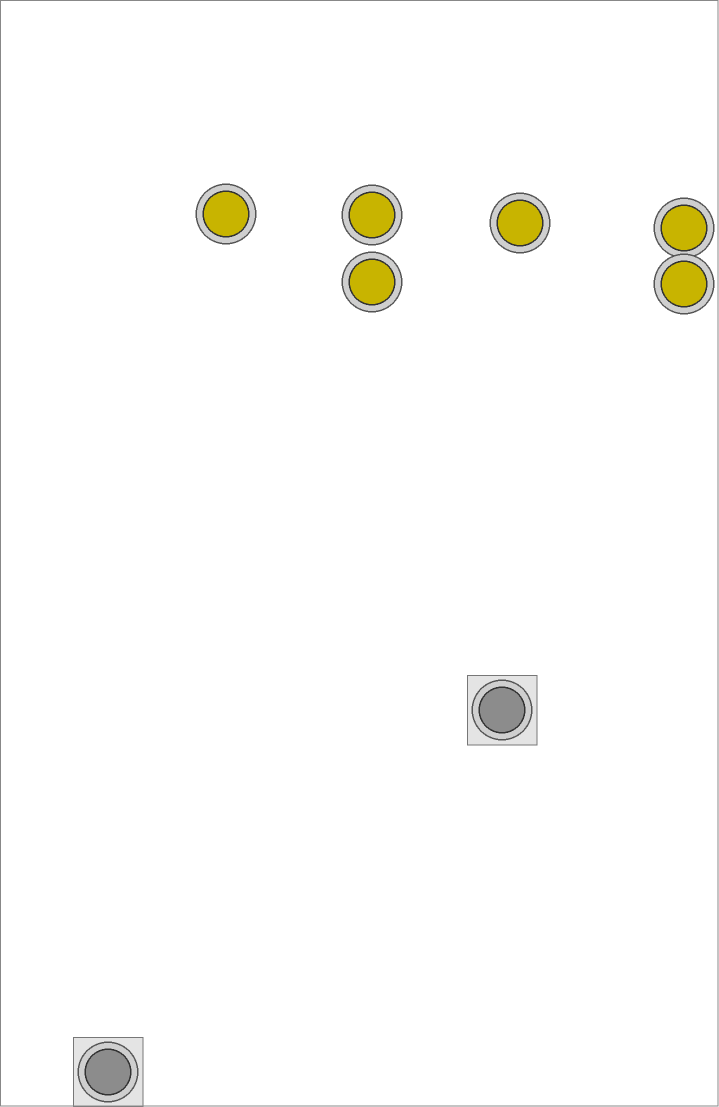
VISUALIZATION Screen1  // 719x1107
    Lamp1 (191,179 70x70), variable: HMI.led1_1, style: Lamp-Lamp1-Yellow
    Lamp1 (337,247 70x70), variable: HMI.led2_2, style: Lamp-Lamp1-Yellow
    Lamp1 (337,180 70x70), variable: HMI.led2_1, style: Lamp-Lamp1-Yellow
    Lamp1 (485,188 70x70), variable: HMI.led3, style: Lamp-Lamp1-Yellow
    Lamp1 (649,193 70x70), variable: HMI.led4_1, style: Lamp-Lamp1-Yellow
    Lamp1 (649,249 70x70), variable: HMI.led4_2, style: Lamp-Lamp1-Yellow
    PushSwitch (467,675 70x70), variable: HMI.btn, behaviour: TAP, style: Switch-PushSwitch-Gray
    PushSwitch (73,1037 70x70), variable: MAIN.isDay, behaviour: TOGGLE, style: Switch-PushSwitch-Gray
END_VISUALIZATION
